(* CODESYS project SPT_Base_Types.library
   Company: Beckhoff Automation LLC
   DefaultNamespace: SPT_BaseTypes
   Version: 3.2.3
   Placeholder: SPT Base Types
   Title: SPT Base Types

Project tree, tasks and I/O mapping:
  libraries: SPT Event Logger, * (Beckhoff Automation LLC); Tc2_EtherCAT, * (Beckhoff Automation GmbH); Tc2_Standard, * (Beckhoff Automation GmbH); Tc2_System, * (Beckhoff Automation GmbH); Tc2_Utilities, * (Beckhoff Automation GmbH); Tc3_EventLogger, * (Beckhoff Automation GmbH); Tc3_JsonXml, * (Beckhoff Automation GmbH); Tc3_PackML_V2, * (Beckhoff Automation GmbH)
  Component Base/
    HMI/
      data type ST_ComponentBase_Command
      data type ST_ComponentBase_Config
      data type ST_ComponentBase_HMI
      data type ST_ComponentBase_Status
    function block FB_ComponentBase [ST]: AllowHMIControl, BlockHMIControl, Reset, CurrentAlarmSeverity, InSimulation, Name, ParentResponseDefinitions, CyclicLogic, CreateEvents, HMICommunication, Initialize, Monitoring, RaiseAlarm, RaiseAlarmWithStrings, RaiseEventWithStrings
  Framework Base/
    function block FB_BaseFB [ST]: Busy, Error, ErrorID, Marker, Trace, TraceWithJson
    function block FB_CyclicFB [ST]: CyclicLogic, InitComplete
  Interfaces/
    interface I_BaseFB: Busy, Error, ErrorID
    interface I_ComponentBase: AllowHMIControl, BlockHMIControl, Reset, CurrentAlarmSeverity, InSimulation, Name, ParentResponseDefinitions
    interface I_CyclicFB: CyclicLogic, InitComplete
    interface I_PackML_BaseModule: CurrentAlarmSeverity, LogModeChanges, LogStateChanges, Name, ParentResponseDefinitions
    interface I_PackML_Control: ChangeMode, ChangeState, CurrentMode, CurrentState, ModeCommand, StateCommand
    interface I_PackML_ExternalController: Control, ModeChanged, StateChanged
  PackML/
    ControlSource/
      function block FB_ControlSource [ST]: CyclicLogic, Control, ModeChanged, StateChanged, Initialize, Registered
      data type ST_PackML_Control
      data type ST_PackML_Control_Simplified
    DUT/
      data type E_AlarmResponse
      data type E_PMLUnitMode
      data type ST_PackML_SubUnitInfoExt
    HMI/
      data type ST_PackMLBaseModule_Command
      data type ST_PackMLBaseModule_Config
      data type ST_PackMLBaseModule_HMI
      data type ST_PackMLBaseModule_Status
    function block FB_PackML_BaseModule [ST]: CyclicLogic, CurrentAlarmSeverity, LogModeChanges, LogStateChanges, Name, ParentResponseDefinitions, ChangeMode, ChangeState, CurrentMode, CurrentState, ModeCommand, StateCommand, AbortImmediate, AbortImmediateError, HoldControlled, HoldImmediate, StopControlled, StopImmediate, SuspendControlled, SuspendImmediate, RaiseAlarmWithStrings, AllowHMIControl, BlockHMIControl, HMICommunication, HMIPermissions, ComponentMonitor, SubModuleMonitor, Aborted, Complete, Execute, Held, Idle, Stopped, Suspended, Undefined, ModeControl, StateControl, Aborting, Clearing, Completing, Holding, Resetting, Starting, Stopping, Suspending, Unholding, Unsuspending, CreateEvents, Initialize, RegisterComponent, RegisterExternalController, RegisterSubmodule, StateComplete
    function block FB_PackML_ModeLogger [ST]
    function block FB_PackML_StateLogger [ST]
  Project Information/
    function F_GetCompany [ST]
    function F_GetTitle [ST]
    function F_GetVersion [ST]
  Tracing/
    function block FB_TraceLog [ST]: AddContext, AddEntry, AddEntryWithJson, FB_init, TracingAllowed
    global variables Tracing
  Version/
    global variables Global_Version
  VISUs/
    visualisation V_MachineModule
    visualisation V_Module
  text list GlobalTextList
  00000000-0000-0000-0000-000000000000|LICENSE
  LICENSE
  global variables Parameters_BaseComponent
  global variables Parameters_PackML_Base
  global variables Parameters_Tracing
*)

// Component Base/HMI/ST_ComponentBase_Command
TYPE ST_ComponentBase_Command :
	STRUCT
		SimulatedOperation : BOOL;
		StandardOperation  : BOOL;
		Reset			   : BOOL;
	END_STRUCT
END_TYPE

// Component Base/HMI/ST_ComponentBase_Config
TYPE ST_ComponentBase_Config :
	STRUCT
		Name : STRING;
	END_STRUCT
END_TYPE

// Component Base/HMI/ST_ComponentBase_HMI
TYPE ST_ComponentBase_HMI :
	STRUCT
		Config	: ST_ComponentBase_Config;
		Command : ST_ComponentBase_Command;
		Status	: ST_ComponentBase_Status;
	END_STRUCT
END_TYPE

// Component Base/HMI/ST_ComponentBase_Status
TYPE ST_ComponentBase_Status :
	STRUCT
		InSimulation		: BOOL;
		Busy				: BOOL;
		Error				: BOOL;
		ErrorID				: UDINT;
		HMIControlAvailable : BOOL; //Set TRUE *FROM PLC* when HMI requests can be processed
	END_STRUCT
END_TYPE

// PackML/ControlSource/ST_PackML_Control
TYPE ST_PackML_Control :
	STRUCT
		CurrentMode		 : E_PMLUnitMode;
		ModeCommand		 : E_PMLUnitMode;
		CurrentState	 : E_PMLState;
		StateCommand	 : E_PMLCommand;
		ModeNames		 : ARRAY[0..31] OF STRING;
		ModeCommandLast	 : E_PMLUnitMode;
		StateCommandLast : E_PMLCommand;
	END_STRUCT
END_TYPE

// PackML/ControlSource/ST_PackML_Control_Simplified
TYPE ST_PackML_Control_Simplified :
	STRUCT
		ResetPermissive		: BOOL;
		StartPermissive		: BOOL;
		StopPermissive		: BOOL;
		ResetPressed AT %I* : BOOL;
		StartPressed AT %I* : BOOL;
		StopPressed	 AT %I* : BOOL;
	END_STRUCT
END_TYPE

// PackML/DUT/E_AlarmResponse
//! @summary Defines the reaction behavior to a fault
{attribute 'qualified_only'}
{attribute 'strict'}
TYPE E_AlarmResponse : (
		Abort_ImmediateError,
		Abort_Immediate,
		Stop_Immediate,
		Stop_Controlled,
		Hold_Immediate,
		Hold_Controlled,
		Suspend_Immediate,
		Suspend_Controlled,
		NoResponse
	);
END_TYPE

// PackML/DUT/E_PMLUnitMode
//! @summary Defines the allowable PackML modes  
TYPE E_PMLUnitMode : (
		ePMLUnitMode_Invalid	 := 0,
		ePMLUnitMode_Production	 := 1,
		ePMLUnitMode_Maintenance := 2,
		ePMLUnitMode_Manual		 := 3,
		ePMLUnitMode_UserMode1	 := 4,
		ePMLUnitMode_UserMode2	 := 5,
		ePMLUnitMode_UserMode3	 := 6,
		ePMLUnitMode_UserMode4	 := 7,
		ePMLUnitMode_UserMode5	 := 8,
		ePMLUnitMode_UserMode6	 := 9,
		ePMLUnitMode_UserMode7	 := 10,
		ePMLUnitMode_UserMode8	 := 11,
		ePMLUnitMode_UserMode9	 := 12,
		ePMLUnitMode_UserMode10	 := 13,
		ePMLUnitMode_UserMode11	 := 14,
		ePMLUnitMode_UserMode12	 := 15,
		ePMLUnitMode_UserMode13	 := 16,
		ePMLUnitMode_UserMode14	 := 17,
		ePMLUnitMode_UserMode15	 := 18,
		ePMLUnitMode_UserMode16	 := 19,
		ePMLUnitMode_UserMode17	 := 20,
		ePMLUnitMode_UserMode18	 := 21,
		ePMLUnitMode_UserMode19	 := 22,
		ePMLUnitMode_UserMode20	 := 23,
		ePMLUnitMode_UserMode21	 := 24,
		ePMLUnitMode_UserMode22	 := 25,
		ePMLUnitMode_UserMode23	 := 26,
		ePMLUnitMode_UserMode24	 := 27,
		ePMLUnitMode_UserMode25	 := 28,
		ePMLUnitMode_UserMode26	 := 29,
		ePMLUnitMode_UserMode27	 := 30,
		ePMLUnitMode_UserMode28	 := 31
	) DINT;
END_TYPE

// PackML/DUT/ST_PackML_SubUnitInfoExt
TYPE ST_PackML_SubUnitInfoExt EXTENDS ST_PMLSubUnitInfo : //Extended Struct of ST_PMLSubUnitInfo
	STRUCT
		ModuleID		: DINT;	  //Machine ID for messaging and Identification
		ModuleName		: STRING; //Human readable machine name for messaging
		UnitModeCurrent : E_PMLProtectedUnitMode;
		ActiveAlarm		: BOOL;
	END_STRUCT
END_TYPE

// PackML/HMI/ST_PackMLBaseModule_Command
TYPE ST_PackMLBaseModule_Command :
	STRUCT
		Mode			   : E_PMLUnitMode				:= Parameters_PackML_Base.UNIT_MODE_DEFAULT;
		State			   : Tc3_PackML_V2.E_PMLCommand := Parameters_PackML_Base.UNIT_STATE_DEFAULT;
		ActivateStateLog   : BOOL; //HMI requests to enable the module
		DeactivateStateLog : BOOL; //HMI requests to disable the module
		ActivateModeLog	   : BOOL; //HMI requests to enable the module
		DeactivatModeLog   : BOOL; //HMI requests to disable the module
	END_STRUCT
END_TYPE

// PackML/HMI/ST_PackMLBaseModule_Config
TYPE ST_PackMLBaseModule_Config :
	STRUCT
		Name			: STRING;		//Human-readable module name for user-side messaging
		LogStateChanges : BOOL := TRUE; //Toggle to permit or suppress state change logging (Should be tied to HMI setting to optionally reduce event logger clutter)
		LogModeChanges	: BOOL := TRUE; //Toggle to permit or suppress state change logging (Should be tied to HMI setting to optionally reduce event logger clutter)
		ModeNames		: ARRAY[0..31] OF STRING;
	END_STRUCT
END_TYPE

// PackML/HMI/ST_PackMLBaseModule_HMI
TYPE ST_PackMLBaseModule_HMI :
	STRUCT
		Config	: ST_PackMLBaseModule_Config;
		Command : ST_PackMLBaseModule_Command;
		Status	: ST_PackMLBaseModule_Status;
	END_STRUCT
END_TYPE

// PackML/HMI/ST_PackMLBaseModule_Status
TYPE ST_PackMLBaseModule_Status :
	STRUCT
		Busy				: BOOL;
		Error				: BOOL;
		ErrorID				: UDINT;
		Mode				: E_PMLUnitMode;
		State				: Tc3_PackML_V2.E_PMLState;
		HMIControlAvailable : BOOL;
	END_STRUCT
END_TYPE

// Tracing/Tracing
{attribute 'qualified_only'}
VAR_GLOBAL
	GlobalTraceLog : FB_TraceLog;
END_VAR

// Version/Global_Version
{attribute 'TcGenerated'}
{attribute 'no-analysis'}
{attribute 'linkalways'}
// This function has been automatically generated from the project information.
VAR_GLOBAL CONSTANT
	{attribute 'const_non_replaced'}
	stLibVersion_SPT_Base_Types : ST_LibVersion := (iMajor := 3, iMinor := 2, iBuild := 3, iRevision := 0, nFlags := 1, sVersion := '3.2.3');
END_VAR

// Parameters_BaseComponent
{attribute 'qualified_only'}
VAR_GLOBAL CONSTANT
	COMPONENT_BASE_ALARM_COUNT : UINT := 2;
END_VAR

// Parameters_PackML_Base
{attribute 'qualified_only'}
VAR_GLOBAL CONSTANT
	MAX_NO_OF_SUBMODULES		   : UDINT						:= 20;
	MAX_NO_OF_COMPONENTS		   : UDINT						:= 32;
	MAX_NO_OF_EXTERNAL_CONTROLLERS : UDINT						:= 10;
	UNIT_MODE_DEFAULT			   : E_PMLUnitMode				:= E_PMLUnitMode.ePMLUnitMode_Production;
	UNIT_STATE_DEFAULT			   : Tc3_PackML_V2.E_PMLCommand := E_PMLCommand.ePMLCommand_Abort;
END_VAR

// Parameters_Tracing
{attribute 'qualified_only'}
VAR_GLOBAL CONSTANT
	TRACING_ENABLED						: BOOL	:= TRUE;
	MAX_LOG_ENTRIES_PER_SCAN			: UDINT := 100;
	ALLOW_DUPLICATE_SEQUENTIAL_MESSAGES : BOOL	:= FALSE;
END_VAR

// Component Base/FB_ComponentBase
//! @summary Basic framework of a component
FUNCTION_BLOCK ABSTRACT FB_ComponentBase EXTENDS FB_CyclicFB IMPLEMENTS I_ComponentBase
VAR
	//I_BasicComponent internal property variables
	_CurrentAlarmSeverity			: TcEventSeverity;
	_Name							: STRING; //String name of the component
	_ParentFaultResponseDefinitions : ARRAY[0..4] OF E_AlarmResponse
		:= [E_AlarmResponse.NoResponse, E_AlarmResponse.NoResponse, E_AlarmResponse.NoResponse, E_AlarmResponse.Abort_ImmediateError, E_AlarmResponse.Abort_ImmediateError];
	_Simulate : BOOL; //TRUE disables all hardware I/O and simulates input and output behavior

	//Alarming
	ComponentBaseAlarms : ARRAY[1..Parameters_BaseComponent.COMPONENT_BASE_ALARM_COUNT] OF FB_TcAlarm;

	//HMI Monitoring and control structure
	ComponentBase_HMI			: ST_ComponentBase_HMI;
	HMICommand_RT				: R_TRIG;
	HMICommandActive_Base		: BOOL;
	HMICommandActive_Descendant : BOOL;
END_VAR

//! @summary Sets permissive bit to allow HMI control of component functions
METHOD PUBLIC AllowHMIControl

//! @description This method is called as required by the parent module of this component
ComponentBase_HMI.Status.HMIControlAvailable := TRUE;
END_METHOD

//! @summary Clears permissive bit to allow HMI control of component functions
METHOD PUBLIC BlockHMIControl

//! @description This method is called as required by the parent module of this component
ComponentBase_HMI.Status.HMIControlAvailable := FALSE;
END_METHOD

//! @summary Clears error flags and error IDs for this component
METHOD PUBLIC Reset : BOOL
//This may or may not be called depending on the component type 

//which derives FB_ComponentBase
F_ClearAllEventsInClass(ComponentBaseAlarms);
Reset := TRUE;
END_METHOD

//! @summary Returns the current alarm severity for this component
PROPERTY CurrentAlarmSeverity : TcEventSeverity
GET
CurrentAlarmSeverity := _CurrentAlarmSeverity;
END_GET
END_PROPERTY

//! @summary Enable/Disable simulation logic for this component
PROPERTY InSimulation : BOOL
GET
InSimulation := _Simulate;
END_GET
SET
_Simulate := InSimulation;
END_SET
END_PROPERTY

//! @summary Get/Set this component's name
PROPERTY Name : STRING
GET
Name := _Name;
END_GET
SET
_Name := Name;
END_SET
END_PROPERTY

PROPERTY ParentResponseDefinitions : ARRAY[0..4] OF E_AlarmResponse
GET
ParentResponseDefinitions[TcEventSeverity.Verbose]	:= _ParentFaultResponseDefinitions[TcEventSeverity.Verbose];
ParentResponseDefinitions[TcEventSeverity.Info]		:= _ParentFaultResponseDefinitions[TcEventSeverity.Info];
ParentResponseDefinitions[TcEventSeverity.Warning]	:= _ParentFaultResponseDefinitions[TcEventSeverity.Warning];
ParentResponseDefinitions[TcEventSeverity.Error]	:= _ParentFaultResponseDefinitions[TcEventSeverity.Error];
ParentResponseDefinitions[TcEventSeverity.Critical] := _ParentFaultResponseDefinitions[TcEventSeverity.Critical];
END_GET
SET
_ParentFaultResponseDefinitions[TcEventSeverity.Verbose]  := ParentResponseDefinitions[TcEventSeverity.Verbose];
_ParentFaultResponseDefinitions[TcEventSeverity.Info]	  := ParentResponseDefinitions[TcEventSeverity.Info];
_ParentFaultResponseDefinitions[TcEventSeverity.Warning]  := ParentResponseDefinitions[TcEventSeverity.Warning];
_ParentFaultResponseDefinitions[TcEventSeverity.Error]	  := ParentResponseDefinitions[TcEventSeverity.Error];
_ParentFaultResponseDefinitions[TcEventSeverity.Critical] := ParentResponseDefinitions[TcEventSeverity.Critical];
END_SET
END_PROPERTY

//! @summary This method serves as the entry point for all underlying FB logic
METHOD PUBLIC CyclicLogic

//! @description This method should be called cyclically by descendant function blocks by invoking <c>SUPER^.CyclicLogic()</c>.  Alternatively, the contents of this method could be reimplemented entirely in which case a call to this method would not be necessary.
IF NOT _InitComplete THEN
	_InitComplete := Initialize();
	RETURN;
END_IF

Monitoring();		//Constant error and status monitoring
HMICommunication(); //Keeps the HMI data up to date, and processes requests from the HMI for this component
END_METHOD

//! @summary Initializes event function blocks using this components's name
{attribute 'call_after_online_change_slot' := '<slot>'}
METHOD PROTECTED CreateEvents

//! @description This method is called by <c>Initialize()</c> as required
F_CreateAllEventsInClass(Alarms		:= ComponentBaseAlarms,
						 ClassSize	:= SIZEOF(TC_EVENTS.ComponentBase),
						 pInitEvent := ADR(TC_EVENTS.ComponentBase.InitReferenceEvent),
						 Prefix		:= _Name);
END_METHOD

//! @summary Provides interlocks for HMI control and updates HMI status information for this component
METHOD PROTECTED HMICommunication

//! @description This method is called cyclically by <c>CyclicLogic()</c>
//Extend this method in extended FBs to communicate specific implementation data

//Process HMI requests
HMICommand_RT(CLK := (ComponentBase_HMI.Status.HMIControlAvailable AND NOT HMICommandActive_Descendant) AND
					 (ComponentBase_HMI.Command.Reset XOR ComponentBase_HMI.Command.SimulatedOperation XOR ComponentBase_HMI.Command.StandardOperation));

//Desendant components should observe this to interlock HMI commands
HMICommandActive_Base :=
	ComponentBase_HMI.Status.HMIControlAvailable AND (ComponentBase_HMI.Command.Reset OR ComponentBase_HMI.Command.SimulatedOperation OR ComponentBase_HMI.Command.StandardOperation);

IF HMICommand_RT.Q THEN
	IF ComponentBase_HMI.Command.Reset THEN
		Reset();
	END_IF

	IF ComponentBase_HMI.Command.SimulatedOperation THEN
		_Simulate := TRUE;
	END_IF

	IF ComponentBase_HMI.Command.StandardOperation THEN
		_Simulate := FALSE;
	END_IF
END_IF

//Update HMI status info
ComponentBase_HMI.Config.Name		  := _Name;
ComponentBase_HMI.Status.Busy		  := _Busy;
ComponentBase_HMI.Status.Error		  := _Error;
ComponentBase_HMI.Status.InSimulation := _Simulate;
ComponentBase_HMI.Status.ErrorID	  := _ErrorID;
END_METHOD

//! @summary Basic component initialization logic
METHOD PROTECTED Initialize : BOOL;

//! @description This method is called by <c>CyclicLogic()</c> as required
//Extend initialize as needed in extended FBs
CreateEvents();
Initialize := TRUE;
END_METHOD

//! Provides basic error detection and event handling for this component
METHOD PROTECTED Monitoring

(*! @descriptionThis method is called cyclically by <c>CyclicLogic()</c>*)
//Extend from extended FB with monitoring logic
IF NOT ComponentBaseAlarms[E_ComponentBase.SimulationWarning].bRaised AND _Simulate THEN
	ComponentBaseAlarms[E_ComponentBase.SimulationWarning].Raise(0);
ELSIF ComponentBaseAlarms[E_ComponentBase.SimulationWarning].bRaised AND NOT _Simulate THEN
	ComponentBaseAlarms[E_ComponentBase.SimulationWarning].Clear(0, 0);
END_IF

_CurrentAlarmSeverity := TcEventSeverity.Verbose;
_CurrentAlarmSeverity := F_GetMaxSeverityRaised(Alarms := ComponentBaseAlarms, CurrentSeverity := _CurrentAlarmSeverity);
END_METHOD

//! @summary Raise an alarm, passing the faulted FB's error ID as a paramter
METHOD PROTECTED RaiseAlarm
VAR_IN_OUT
	Alarm : FB_TcAlarm;
END_VAR
F_RaiseAlarm(Alarm := Alarm);
END_METHOD

//! @summary Raises an alarm and passes string arguments as parameters for extra fault context/info
METHOD PROTECTED RaiseAlarmWithStrings
VAR_IN_OUT
	Alarm : FB_TcAlarm; //! Alarm to be raised
END_VAR

VAR_INPUT
	String_1 : STRING; //! First string parameter (The Name of this component will be applied first automatically)
	String_2 : STRING; //! Second string parameter
END_VAR
F_RaiseAlarmWithStringsAndFlags(Alarm	  := Alarm,
								ErrorFlag := _Error,
								ErrorID	  := _ErrorID,
								String_1  := _Name,
								String_2  := String_1,
								String_3  := String_2);
END_METHOD

//! @summary Raises an alarm and passes string arguments as parameters for extra fault context/info
METHOD PROTECTED RaiseEventWithStrings
VAR_IN_OUT
	Alarm : FB_TcAlarm; //! Alarm to be raised
END_VAR

VAR_INPUT
	String_1 : STRING; //! First string parameter (The Name of this component will be applied first automatically)
	String_2 : STRING; //! Second string parameter
END_VAR
F_RaiseAlarmWithStringParameters(Alarm	  := Alarm,
								 String_1 := _Name,
								 String_2 := String_1,
								 String_3 := String_2);
END_METHOD

END_FUNCTION_BLOCK

// Framework Base/FB_CyclicFB
FUNCTION_BLOCK ABSTRACT FB_CyclicFB EXTENDS FB_BaseFB IMPLEMENTS I_CyclicFB
VAR
	_InitComplete : BOOL;
END_VAR

// Derivatives of FB_CyclicFB should *NOT* have code in the function block body

// Use CyclicLogic() instead

METHOD PUBLIC ABSTRACT CyclicLogic
VAR_INPUT
END_VAR
END_METHOD

PROPERTY InitComplete : BOOL
GET
InitComplete := _InitComplete;
END_GET
END_PROPERTY

END_FUNCTION_BLOCK

// Framework Base/FB_BaseFB
{attribute 'reflection'}
FUNCTION_BLOCK ABSTRACT FB_BaseFB IMPLEMENTS I_BaseFB
VAR
	{attribute 'instance-path'}
	{attribute 'noinit'}
	InstancePath : STRING;
END_VAR

// I_BaseFB
VAR
	_Busy	 : BOOL := TRUE;
	_Error	 : BOOL;
	_ErrorID : UDINT;
END_VAR

// Derivatives of FB_BaseFB can have code in the function block body

PROPERTY Busy : BOOL
GET
Busy := _Busy;
END_GET
END_PROPERTY

PROPERTY Error : BOOL
GET
Error := _Error;
END_GET
END_PROPERTY

PROPERTY ErrorID : UDINT
GET
ErrorID := _ErrorID;
END_GET
END_PROPERTY

METHOD PUBLIC Marker
VAR_INPUT
	Message : T_MaxString;
END_VAR
Tracing.GlobalTraceLog.AddEntry(InstancePath, Message, 1);
END_METHOD

METHOD PUBLIC Trace
VAR_INPUT
	Message : T_MaxString;
END_VAR
Tracing.GlobalTraceLog.AddEntry(InstancePath, Message, 0);
END_METHOD

METHOD PUBLIC TraceWithJson
VAR_INPUT
	Message : T_MaxString;
	Json	: T_MaxString;
END_VAR
Tracing.GlobalTraceLog.AddEntryWithJson(InstancePath,
										Message,
										0,
										Json);
END_METHOD

END_FUNCTION_BLOCK

// Interfaces/I_BaseFB
INTERFACE I_BaseFB EXTENDS __SYSTEM.IQueryInterface

PROPERTY Busy : BOOL
GET
END_GET
END_PROPERTY

PROPERTY Error : BOOL
GET
END_GET
END_PROPERTY

PROPERTY ErrorID : UDINT;
GET
END_GET
END_PROPERTY

END_INTERFACE

// Interfaces/I_CyclicFB
INTERFACE I_CyclicFB EXTENDS I_BaseFB

METHOD CyclicLogic
VAR_INPUT
END_VAR
END_METHOD

PROPERTY InitComplete : BOOL
GET
END_GET
END_PROPERTY

END_INTERFACE

// Interfaces/I_ComponentBase
INTERFACE I_ComponentBase EXTENDS I_CyclicFB

METHOD PUBLIC AllowHMIControl
VAR_INPUT
END_VAR
END_METHOD

METHOD PUBLIC BlockHMIControl
VAR_INPUT
END_VAR
END_METHOD

METHOD PUBLIC Reset : BOOL
END_METHOD

PROPERTY CurrentAlarmSeverity : TcEventSeverity
GET
END_GET
END_PROPERTY

PROPERTY InSimulation : BOOL
GET
END_GET
SET
END_SET
END_PROPERTY

PROPERTY Name : STRING
GET
END_GET
SET
END_SET
END_PROPERTY

PROPERTY ParentResponseDefinitions : ARRAY[0..4] OF E_AlarmResponse
GET
END_GET
SET
END_SET
END_PROPERTY

END_INTERFACE

// Interfaces/I_PackML_BaseModule
INTERFACE I_PackML_BaseModule EXTENDS I_CyclicFB, I_PackML_Control

PROPERTY CurrentAlarmSeverity : TcEventSeverity
GET
END_GET
END_PROPERTY

PROPERTY LogModeChanges : BOOL
GET
END_GET
SET
END_SET
END_PROPERTY

PROPERTY LogStateChanges : BOOL
GET
END_GET
SET
END_SET
END_PROPERTY

PROPERTY Name : STRING
GET
END_GET
SET
END_SET
END_PROPERTY

PROPERTY ParentResponseDefinitions : ARRAY[0..4] OF E_AlarmResponse
GET
END_GET
SET
END_SET
END_PROPERTY

END_INTERFACE

// Interfaces/I_PackML_Control
INTERFACE I_PackML_Control

METHOD ChangeMode
VAR_INPUT
	Mode : E_PMLUnitMode;
END_VAR
END_METHOD

METHOD ChangeState
VAR_INPUT
	State : E_PMLCommand;
END_VAR
END_METHOD

PROPERTY CurrentMode : E_PMLUnitMode
GET
END_GET
END_PROPERTY

PROPERTY CurrentState : E_PMLState
GET
END_GET
END_PROPERTY

PROPERTY ModeCommand : DINT
GET
END_GET
SET
END_SET
END_PROPERTY

PROPERTY StateCommand : E_PMLCommand
GET
END_GET
SET
END_SET
END_PROPERTY

END_INTERFACE

// Interfaces/I_PackML_ExternalController
INTERFACE I_PackML_ExternalController

PROPERTY Control : I_PackML_Control
SET
END_SET
END_PROPERTY

METHOD ModeChanged
VAR_INPUT
	NewMode : E_PMLUnitMode;
END_VAR
END_METHOD

METHOD StateChanged
VAR_INPUT
	NewState : E_PMLCommand;
END_VAR
END_METHOD

END_INTERFACE

// PackML/ControlSource/FB_ControlSource
FUNCTION_BLOCK FB_ControlSource EXTENDS FB_CyclicFB IMPLEMENTS I_PackML_ExternalController
VAR
	ipModule				  : I_PackML_Control;
	MainPMLControl_Simplified : ST_PackML_Control_Simplified;
	MainPMLControl_Standard	  : ST_PackML_Control;
	R_HMICommand			  : R_TRIG;
END_VAR

METHOD CyclicLogic
VAR
	i : UDINT;
END_VAR
IF NOT _InitComplete THEN
	_InitComplete := Initialize();
	RETURN;
END_IF

//Copy the module to the local mode and state
MainPMLControl_Standard.CurrentMode	 := ipModule.CurrentMode;
MainPMLControl_Standard.CurrentState := ipModule.CurrentState;
FOR i := 1 TO 5 DO
	MainPMLControl_Standard.ModeNames[i] := F_UnitModeToString(TO_DINT(i));
END_FOR

//Process requests
R_HMICommand(CLK := (MainPMLControl_Simplified.ResetPressed XOR MainPMLControl_Simplified.StartPressed XOR MainPMLControl_Simplified.StopPressed) XOR
					(MainPMLControl_Standard.StateCommand <> E_PMLCommand.ePMLCommand_Undefined AND MainPMLControl_Standard.StateCommandLast <> MainPMLControl_Standard.StateCommand) XOR
					(MainPMLControl_Standard.ModeCommandLast <> MainPMLControl_Standard.ModeCommand));

IF R_HMICommand.Q THEN
	MainPMLControl_Standard.ModeCommandLast	 := MainPMLControl_Standard.ModeCommand;
	MainPMLControl_Standard.StateCommandLast := MainPMLControl_Standard.StateCommand;
	IF MainPMLControl_Simplified.ResetPressed AND MainPMLControl_Simplified.ResetPermissive AND MainPMLControl_Standard.CurrentState = E_PMLState.ePMLState_Aborted THEN
		ipModule.ChangeState(Tc3_PackML_V2.E_PMLCommand.ePMLCommand_Clear);
	ELSIF MainPMLControl_Simplified.ResetPressed AND MainPMLControl_Simplified.ResetPermissive THEN
		ipModule.ChangeState(Tc3_PackML_V2.E_PMLCommand.ePMLCommand_Reset);
	ELSIF MainPMLControl_Simplified.StartPressed AND MainPMLControl_Simplified.StartPermissive THEN
		IF MainPMLControl_Standard.CurrentState = Tc3_PackML_V2.E_PMLState.ePMLState_Idle THEN
			ipModule.ChangeState(Tc3_PackML_V2.E_PMLCommand.ePMLCommand_Start);
		ELSIF MainPMLControl_Standard.CurrentState = Tc3_PackML_V2.E_PMLState.ePMLState_Held THEN
			ipModule.ChangeState(Tc3_PackML_V2.E_PMLCommand.ePMLCommand_Unhold);
		END_IF
	ELSIF MainPMLControl_Simplified.StopPressed AND MainPMLControl_Simplified.StopPermissive THEN
		ipModule.ChangeState(Tc3_PackML_V2.E_PMLCommand.ePMLCommand_Stop);
	ELSIF ipModule.StateCommand <> MainPMLControl_Standard.StateCommand THEN
		ipModule.StateCommand := MainPMLControl_Standard.StateCommand;
	ELSIF ipModule.ModeCommand <> MainPMLControl_Standard.ModeCommand THEN
		ipModule.ModeCommand := MainPMLControl_Standard.ModeCommand;
	END_IF
END_IF

//Set the permissives for each button
MainPMLControl_Simplified.StartPermissive :=
	MainPMLControl_Standard.CurrentState = Tc3_PackML_V2.E_PMLState.ePMLState_Idle OR MainPMLControl_Standard.CurrentState = Tc3_PackML_V2.E_PMLState.ePMLState_Held;

MainPMLControl_Simplified.StopPermissive :=
	(MainPMLControl_Standard.CurrentState <> Tc3_PackML_V2.E_PMLState.ePMLState_Stopped AND MainPMLControl_Standard.CurrentState <> Tc3_PackML_V2.E_PMLState.ePMLState_Clearing AND
	 MainPMLControl_Standard.CurrentState <> Tc3_PackML_V2.E_PMLState.ePMLState_Aborted AND MainPMLControl_Standard.CurrentState <> Tc3_PackML_V2.E_PMLState.ePMLState_Aborting AND
	 MainPMLControl_Standard.CurrentState <> Tc3_PackML_V2.E_PMLState.ePMLState_Idle AND MainPMLControl_Standard.CurrentState <> Tc3_PackML_V2.E_PMLState.ePMLState_Undefined);

MainPMLControl_Simplified.ResetPermissive :=
	MainPMLControl_Standard.CurrentState = Tc3_PackML_V2.E_PMLState.ePMLState_Complete OR MainPMLControl_Standard.CurrentState = Tc3_PackML_V2.E_PMLState.ePMLState_Stopped OR
	MainPMLControl_Standard.CurrentState = Tc3_PackML_V2.E_PMLState.ePMLState_Aborted;
END_METHOD

PROPERTY Control : I_PackML_Control
SET
ipModule := Control;
END_SET
END_PROPERTY

METHOD FINAL ModeChanged
VAR_INPUT
	NewMode : E_PMLUnitMode;
END_VAR
MainPMLControl_Standard.ModeCommand := NewMode;
END_METHOD

METHOD FINAL StateChanged
VAR_INPUT
	NewState : E_PMLCommand;
END_VAR
MainPMLControl_Standard.StateCommand := NewState;
END_METHOD

METHOD FINAL Initialize : BOOL
IF Registered THEN
	Initialize := TRUE;
END_IF
END_METHOD

PROPERTY Registered : BOOL
GET
Registered := ipModule <> 0;
END_GET
END_PROPERTY

END_FUNCTION_BLOCK

// PackML/FB_PackML_BaseModule
FUNCTION_BLOCK ABSTRACT FB_PackML_BaseModule EXTENDS FB_CyclicFB IMPLEMENTS I_PackML_BaseModule, I_PackML_Control
	//I_PMLControl
VAR
	_CurrentMode	: E_PMLUnitMode; //Current UnitMode of the module	
	_CommandedMode	: E_PMLUnitMode; //Current Commanded UnitMode of the module
	_CurrentState	: Tc3_PackML_V2.E_PMLState;
	_CommandedState : Tc3_PackML_V2.E_PMLCommand;
END_VAR

//I_PMLModuleBase
VAR
	_CurrentAlarmSeverity			: TcEventSeverity;
	_LogModeChanges					: BOOL := TRUE;	 //Toggle to permit or suppress state change logging (Should be tied to HMI setting to optionally reduce event logger clutter)
	_LogStateChanges				: BOOL := FALSE; //Toggle to permit or suppress state change logging (Should be tied to HMI setting to optionally reduce event logger clutter)
	_Name							: STRING;		 //Human-readable module name for user-side messaging
	_ParentFaultResponseDefinitions : ARRAY[0..4] OF E_AlarmResponse
		:= [E_AlarmResponse.NoResponse, E_AlarmResponse.NoResponse, E_AlarmResponse.NoResponse, E_AlarmResponse.Abort_ImmediateError, E_AlarmResponse.Abort_ImmediateError];
END_VAR

VAR
	ModeManager						  : PML_UnitModeManager;		//Manages operating mode transitions and rules
	StateMachine					  : PML_StateMachine;			//Manages PackML state transitions
	CustomModes						  : PML_UnitModeConfig;			//Used to define custom machine modes if desired
	PMLStateLogger					  : FB_PackML_StateLogger;		//Logs PackML state changes
	PMLModeLogger					  : FB_PackML_ModeLogger;		//Logs PackML Mode changes	
	PackMLBaseModule_HMI			  : ST_PackMLBaseModule_HMI;	//Handles status and control communications with the HMI
	PMLSubModuleInfoRef				  : ST_PMLSubUnitInfoRef;		// Reference to the subunit information, used by the state machine
	LastModeCommand					  : E_PMLUnitMode;				//Previous received PackML mode command
	LastMode						  : DINT;						//Last PackML mode 	
	LastState						  : Tc3_PackML_V2.E_PMLState;	//Last cycle PackML state
	StateTasksComplete				  : BOOL := FALSE;				//All tasks to be performed at this program level are complete
	NoStateTasksToComplete			  : BOOL := TRUE;				//Indicates whether this stateneeds to perform tasks other than commanding its children
	PackMLAlarms					  : ARRAY[1..48] OF FB_TcAlarm; //Array of alarms for PackML state and mode changes that exist in any PackML enabled module
	BaseAlarms						  : ARRAY[1..32] OF FB_TcAlarm; //Array of alarms for general module Alarms				
	ipSubModules					  : ARRAY[1..Parameters_PackML_Base.MAX_NO_OF_SUBMODULES] OF I_PackML_BaseModule;
	PMLSubModuleInfo				  : ARRAY[1..Parameters_PackML_Base.MAX_NO_OF_SUBMODULES] OF ST_PMLSubUnitInfo;
	NumberOfSubModules				  : UDINT := 0; //calculated number of instantiated sub modules
	ipComponents					  : ARRAY[1..Parameters_PackML_Base.MAX_NO_OF_COMPONENTS] OF I_ComponentBase;
	NumberOfComponents				  : UDINT := 0; //calculated number of instantiated components
	ModeNames						  : ARRAY[0..31] OF STRING;
	ipExternalControllers			  : ARRAY[1..Parameters_PackML_Base.MAX_NO_OF_EXTERNAL_CONTROLLERS] OF I_PackML_ExternalController;
	ReachedInitialDefaultStateAndMode : BOOL;
	ModeChangeRequested				  : BOOL;
	SequenceState					  : UDINT;
	DescendantSequenceState			  : UDINT;
	HMICommand_RT					  : R_TRIG;
	HMICommandActive_Base			  : BOOL;
	HMICommandActive_Descendant		  : BOOL;
END_VAR

//*********************************************************

// !!!!! Code implementation only in CyclicLogic() method !!!!! 

//*********************************************************

//! @summary This method serves as the entry point for all underlying FB logic

//! @description This method should be called cyclically by descendant function blocks by invoking <c>SUPER^.CyclicLogic()</c>.  Alternatively, the contents of this method could be reimplemented entirely in which case a call to this method would not be necessary.
METHOD PUBLIC CyclicLogic
VAR
	i : UDINT;
END_VAR
//*********************************************************

//If you are about to write actual machine implementation code, note that implementation code should exist within an implementation machine module block that extends this machine module base!

//*********************************************************

// Descendents of this FB which override this methods should

// use SUPER^.Initialize()
IF NOT _InitComplete THEN
	_InitComplete := Initialize();
	RETURN;
END_IF

// Inhibit mode & state errors until startup is complete
IF NOT ReachedInitialDefaultStateAndMode AND _CurrentState = E_PMLState.ePMLState_Aborted AND _CurrentMode = Parameters_PackML_Base.UNIT_MODE_DEFAULT THEN
	ReachedInitialDefaultStateAndMode := TRUE;
END_IF

// Call this module's subunits, if any are defined
FOR i := 1 TO NumberOfSubModules DO
	IF ipSubModules[i] <> 0 THEN
		ipSubModules[i].CyclicLogic();
		PMLSubModuleInfo[i].eState := ipSubModules[i].CurrentState; //Reflect the state of the subunits to the state machine of the module		
	END_IF
END_FOR

FOR i := 1 TO NumberOfComponents DO
	IF ipComponents[i] <> 0 THEN
		ipComponents[i].CyclicLogic();
	END_IF
END_FOR

//Handle HMI communications--this must happen before state control!!
HMICommunication();

// Mode control loop of the module
ModeControl();

// State control loop of the module
StateControl();

//VISUCommunication();

//ExternalControl();
SubModuleMonitor();
ComponentMonitor();
HMIPermissions();
_CurrentAlarmSeverity := TcEventSeverity.Verbose;
_CurrentAlarmSeverity := F_GetMaxSeverityRaised(Alarms := PackMLAlarms, CurrentSeverity := _CurrentAlarmSeverity);
_CurrentAlarmSeverity := F_GetMaxSeverityRaised(Alarms := BaseAlarms, CurrentSeverity := _CurrentAlarmSeverity);
END_METHOD

//! @summary Returns the highest severity of any event(s) currently raised 
PROPERTY CurrentAlarmSeverity : TcEventSeverity
GET
CurrentAlarmSeverity := _CurrentAlarmSeverity;
END_GET
END_PROPERTY

//! @summary Enable/Disable logging of mode changes
PROPERTY LogModeChanges : BOOL
GET
LogModeChanges := _LogModeChanges;
END_GET
SET
_LogModeChanges := LogModeChanges;
END_SET
END_PROPERTY

//! @summary Enable/Disable logging of state changes
PROPERTY LogStateChanges : BOOL
GET
LogStateChanges := _LogStateChanges;
END_GET
SET
_LogStateChanges := LogStateChanges;
END_SET
END_PROPERTY

//! @summary Get/Set the name of this module
PROPERTY Name : STRING
GET
Name := _Name;
END_GET
SET
_Name := Name;
END_SET
END_PROPERTY

//! @summary TODO: does this do anything?
PROPERTY ParentResponseDefinitions : ARRAY[0..4] OF E_AlarmResponse
GET
ParentResponseDefinitions[TcEventSeverity.Verbose]	:= _ParentFaultResponseDefinitions[TcEventSeverity.Verbose];
ParentResponseDefinitions[TcEventSeverity.Info]		:= _ParentFaultResponseDefinitions[TcEventSeverity.Info];
ParentResponseDefinitions[TcEventSeverity.Warning]	:= _ParentFaultResponseDefinitions[TcEventSeverity.Warning];
ParentResponseDefinitions[TcEventSeverity.Error]	:= _ParentFaultResponseDefinitions[TcEventSeverity.Error];
ParentResponseDefinitions[TcEventSeverity.Critical] := _ParentFaultResponseDefinitions[TcEventSeverity.Critical];
END_GET
SET
_ParentFaultResponseDefinitions[TcEventSeverity.Verbose]  := ParentResponseDefinitions[TcEventSeverity.Verbose];
_ParentFaultResponseDefinitions[TcEventSeverity.Info]	  := ParentResponseDefinitions[TcEventSeverity.Info];
_ParentFaultResponseDefinitions[TcEventSeverity.Warning]  := ParentResponseDefinitions[TcEventSeverity.Warning];
_ParentFaultResponseDefinitions[TcEventSeverity.Error]	  := ParentResponseDefinitions[TcEventSeverity.Error];
_ParentFaultResponseDefinitions[TcEventSeverity.Critical] := ParentResponseDefinitions[TcEventSeverity.Critical];
END_SET
END_PROPERTY

METHOD ChangeMode
VAR_INPUT
	Mode : E_PMLUnitMode;
END_VAR
IF Mode <> _CommandedMode THEN
	ModeCommand := Mode;
END_IF
END_METHOD

METHOD ChangeState
VAR_INPUT
	State : E_PMLCommand;
END_VAR
IF State <> _CommandedState THEN
	StateCommand := State;
END_IF
END_METHOD

//! @summary Returns the current PackML mode of this module
PROPERTY CurrentMode : E_PMLUnitMode
GET
CurrentMode := _CurrentMode;
END_GET
END_PROPERTY

//! @summary Returns current PackML state of this module
PROPERTY CurrentState : Tc3_PackML_V2.E_PMLState
GET
CurrentState := _CurrentState;
END_GET
END_PROPERTY

//! @summary Sets the requested PackML Mode
PROPERTY ModeCommand : DINT
GET
ModeCommand := _CommandedMode;
END_GET
SET
VAR
	i : UDINT;
END_VAR
IF ModeCommand <> _CommandedMode THEN
	_CommandedMode					  := ModeCommand;
	PackMLBaseModule_HMI.Command.Mode := ModeCommand;

	//Notify external controllers that state has changed	
	FOR i := 1 TO Parameters_PackML_Base.MAX_NO_OF_EXTERNAL_CONTROLLERS DO
		IF ipExternalControllers[i] <> 0 THEN
			ipExternalControllers[i].ModeChanged(_CommandedMode);
		END_IF
	END_FOR

	//ModeChangeRequested := TRUE;
END_IF
END_SET
END_PROPERTY

//! @summary Sets the requested PackML state
PROPERTY StateCommand : Tc3_PackML_V2.E_PMLCommand
GET
StateCommand := _CommandedState;
END_GET
SET
VAR
	i : UDINT;
END_VAR
IF _CurrentMode <> E_PMLUnitMode.ePMLUnitMode_Invalid AND _CurrentState <> E_PMLState.ePMLState_Undefined THEN
	_CommandedState					   := StateCommand;
	PackMLBaseModule_HMI.Command.State := StateCommand;

	//Notify external controllers that state has changed
	FOR i := 1 TO Parameters_PackML_Base.MAX_NO_OF_EXTERNAL_CONTROLLERS DO
		IF ipExternalControllers[i] <> 0 THEN
			ipExternalControllers[i].StateChanged(_CommandedState);
		END_IF
	END_FOR
END_IF
END_SET
END_PROPERTY

//! @summary Provides fault reaction logic where the module state is driven to the <b>Aborting</b> state
METHOD PROTECTED AbortImmediate

//! @description No error is thrown by this fault reaction.

//! @description This method is called by <c>ComponentMonitor()</c> or <c>SubModuleMonitor()</c> as required
ChangeState(E_PMLCommand.ePMLCommand_Abort);
END_METHOD

//! @summary Provides fault reaction logic where the module state is driven to the <b>Aborting</b> state
METHOD PROTECTED AbortImmediateError
VAR_INPUT
	Name	 : STRING; //! The name of the faulting submodule or component
	IsModule : BOOL;   //! If TRUE a SubModuleError is thrown.  If FALSE a ComponentError is thrown. 
END_VAR

//! @description This fault reaction throws an accompanying error

//! @description This method is called by <c>ComponentMonitor()</c> or <c>SubModuleMonitor()</c> as required
IF IsModule THEN
	IF NOT BaseAlarms[E_BaseAlarms.SubModuleError].bRaised THEN
		F_RaiseAlarmWithStringParameters(BaseAlarms[E_BaseAlarms.SubModuleError],
										 _Name,
										 '',
										 '');
	END_IF
ELSE
	IF NOT BaseAlarms[E_BaseAlarms.ComponentError].bRaised THEN
		F_RaiseAlarmWithStringParameters(BaseAlarms[E_BaseAlarms.ComponentError],
										 _Name,
										 '',
										 '');
	END_IF
END_IF

THIS^.ChangeState(E_PMLCommand.ePMLCommand_Abort);
END_METHOD

//! @summary Provides fault reaction logic where the module state is driven to the <b>Holding</b> state at the next available opportunity
METHOD PROTECTED HoldControlled

(*! <description> No error is thrown by this fault reaction.
	<b> TODO: Needs implementation </b> </description>*)

//! @description This method is called by <c>ComponentMonitor()</c> or <c>SubModuleMonitor()</c> as required
ChangeState(E_PMLCommand.ePMLCommand_Hold);
END_METHOD

//! @summary Provides fault reaction logic where the module state is driven to the <b>Holding</b> state immediately
METHOD PROTECTED HoldImmediate

(*! <description> No error is thrown by this fault reaction.
	<b> TODO: Needs implementation </b> </description>*)

//! @description This method is called by <c>ComponentMonitor()</c> or <c>SubModuleMonitor()</c> as required
ChangeState(E_PMLCommand.ePMLCommand_Hold);
END_METHOD

//! @summary Provides fault reaction logic where the module state is driven to the <b>Stopping</b> state at the next available opportunity
METHOD PROTECTED StopControlled

(*! <description> No error is thrown by this fault reaction.
	<b> TODO: Needs implementation </b> </description>*)

//! @description This method is called by <c>ComponentMonitor()</c> or <c>SubModuleMonitor()</c> as required
ChangeState(E_PMLCommand.ePMLCommand_Stop);
END_METHOD

//! @summary Provides fault reaction logic where the module state is driven to the <b>Stopping</b> state immediately
METHOD PROTECTED StopImmediate

//! @description No error is thrown by this fault reaction.

//! @description This method is called by <c>ComponentMonitor()</c> or <c>SubModuleMonitor()</c> as required
ChangeState(E_PMLCommand.ePMLCommand_Stop);
END_METHOD

//! @summary Provides fault reaction logic where the module state is driven to the <b>Suspending</b> state at the next available opportunity
METHOD PROTECTED SuspendControlled

(*! <description> No error is thrown by this fault reaction.
	<b> TODO: Needs implementation </b> </description>*)

//! @description This method is called by <c>ComponentMonitor()</c> or <c>SubModuleMonitor()</c> as required
ChangeState(E_PMLCommand.ePMLCommand_Suspend);
END_METHOD

//! @summary Provides fault reaction logic where the module state is driven to the <b>Suspending</b> state immediately
METHOD PROTECTED SuspendImmediate

(*! <description> No error is thrown by this fault reaction.
	<b> TODO: Needs implementation </b> </description>*)

//! @description This method is called by <c>ComponentMonitor()</c> or <c>SubModuleMonitor()</c> as required
ChangeState(E_PMLCommand.ePMLCommand_Suspend);
END_METHOD

//! @summary Raises an alarm and passes string arguments as parameters for extra fault context/info
METHOD PROTECTED RaiseAlarmWithStrings
VAR_IN_OUT
	Alarm : FB_TcAlarm; //! Alarm to be raised
END_VAR

VAR_INPUT
	String_1 : STRING; //! First string parameter (The Name of this component will be applied first automatically)
	String_2 : STRING; //! Second string parameter
END_VAR
F_RaiseAlarmWithStringParameters(Alarm	  := Alarm,
								 String_1 := Name,
								 String_2 := String_1,
								 String_3 := String_2);
END_METHOD

//! @summary Sets permissive bit to allow HMI control of module and component functions
METHOD PROTECTED FINAL AllowHMIControl
VAR_INPUT
	ThisModuleOnly : BOOL; //! If TRUE, only the PackML module itself is controllable. If FALSE, all components become controllable as well
END_VAR

VAR
	i : UDINT;
END_VAR

//! @description This method is called as required by the <c>HMIPermissions()</c> method
PackMLBaseModule_HMI.Status.HMIControlAvailable := TRUE;
IF ThisModuleOnly THEN
	FOR i := 1 TO NumberOfComponents DO
		ipComponents[i].BlockHMIControl();
	END_FOR
ELSE
	FOR i := 1 TO NumberOfComponents DO
		ipComponents[i].AllowHMIControl();
	END_FOR
END_IF
END_METHOD

//! @summary Clears permissive bit to disallow HMI control of module and component functions
METHOD PROTECTED FINAL BlockHMIControl
VAR
	i : UDINT;
END_VAR

//! @description This method is called as required by the <c>HMIPermissions()</c> method
PackMLBaseModule_HMI.Status.HMIControlAvailable := FALSE;
FOR i := 1 TO NumberOfComponents DO
	ipComponents[i].BlockHMIControl();
END_FOR
END_METHOD

//! @summary Provides interlocks for HMI control and updates HMI status information for this module
METHOD PROTECTED HMICommunication

//! @description This method is called cyclically by <c>CyclicLogic()</c>
//Extend this method in extended FBs to communicate specific implementation data

//Process HMI requests
HMICommand_RT(CLK := (PackMLBaseModule_HMI.Status.HMIControlAvailable AND NOT HMICommandActive_Descendant) AND
					 (PackMLBaseModule_HMI.Command.ActivateModeLog XOR PackMLBaseModule_HMI.Command.DeactivatModeLog XOR PackMLBaseModule_HMI.Command.ActivateStateLog XOR
					 PackMLBaseModule_HMI.Command.DeactivateStateLog XOR PackMLBaseModule_HMI.Command.Mode <> _CommandedMode XOR PackMLBaseModule_HMI.Command.State <> _CommandedState));

//Desendant components should observe this to interlock HMI commands
HMICommandActive_Base := PackMLBaseModule_HMI.Status.HMIControlAvailable AND
						 (PackMLBaseModule_HMI.Command.ActivateModeLog OR PackMLBaseModule_HMI.Command.DeactivatModeLog OR PackMLBaseModule_HMI.Command.ActivateStateLog OR
						 PackMLBaseModule_HMI.Command.DeactivateStateLog XOR PackMLBaseModule_HMI.Command.Mode <> _CommandedMode XOR PackMLBaseModule_HMI.Command.State <> _CommandedState);

IF HMICommand_RT.Q THEN
	IF PackMLBaseModule_HMI.Command.ActivateModeLog THEN
		_LogModeChanges := TRUE;
	END_IF

	IF PackMLBaseModule_HMI.Command.DeactivatModeLog THEN
		_LogModeChanges := FALSE;
	END_IF

	IF PackMLBaseModule_HMI.Command.ActivateStateLog THEN
		_LogStateChanges := TRUE;
	END_IF

	IF PackMLBaseModule_HMI.Command.DeactivateStateLog THEN
		_LogStateChanges := FALSE;
	END_IF

	IF PackMLBaseModule_HMI.Command.Mode <> _CommandedMode THEN
		ModeCommand := PackMLBaseModule_HMI.Command.Mode;
	END_IF

	IF PackMLBaseModule_HMI.Command.State <> _CommandedState THEN
		StateCommand := PackMLBaseModule_HMI.Command.State;
	END_IF
END_IF

PackMLBaseModule_HMI.Config.Name			:= _Name;
PackMLBaseModule_HMI.Config.LogModeChanges	:= _LogModeChanges;
PackMLBaseModule_HMI.Config.LogStateChanges := _LogStateChanges;
PackMLBaseModule_HMI.Config.ModeNames		:= ModeNames;
PackMLBaseModule_HMI.Status.Mode			:= _CurrentMode;
PackMLBaseModule_HMI.Status.State			:= _CurrentState;
PackMLBaseModule_HMI.Status.Busy			:= _Busy;
PackMLBaseModule_HMI.Status.Error			:= _Error;
PackMLBaseModule_HMI.Status.ErrorID			:= _ErrorID;
END_METHOD

//! @summary Automatically enables and disables HMI control based on the PackML mode
METHOD PROTECTED HMIPermissions

//! @description This method is called cyclically by <c>CyclicLogic()</c>
//General Mode Based Monitoring and handling of HMI control
CASE _CurrentMode OF
	E_PMLUnitMode.ePMLUnitMode_Production:
		CASE _CurrentState OF
			E_PMLState.ePMLState_Stopped:
				AllowHMIControl(ThisModuleOnly := TRUE); //Allow control for recovery
			E_PMLState.ePMLState_Idle:
				BlockHMIControl();

			E_PMLState.ePMLState_Suspended:
				BlockHMIControl();

			E_PMLState.ePMLState_Execute:
				BlockHMIControl();

			E_PMLState.ePMLState_Aborted:
				AllowHMIControl(ThisModuleOnly := TRUE); //Allow control for recovery
			E_PMLState.ePMLState_Held:
				AllowHMIControl(ThisModuleOnly := TRUE); //Allow control for recovery
			E_PMLState.ePMLState_Complete:
				BlockHMIControl();
		END_CASE

	E_PMLUnitMode.ePMLUnitMode_Manual:
		AllowHMIControl(ThisModuleOnly := FALSE);

	E_PMLUnitMode.ePMLUnitMode_Maintenance:
		AllowHMIControl(ThisModuleOnly := FALSE);
END_CASE
END_METHOD

//! @summary This method monitors <b>components</b> within this PackML module and initiates fault responses as required
METHOD PROTECTED ComponentMonitor : BOOL
VAR
	AlarmResponses : ARRAY[0..4] OF E_AlarmResponse; //Temporary response array
	i			   : UDINT;
END_VAR

//! @description This method is called cyclically by <c>CyclicLogic()</c>
FOR i := 1 TO NumberOfComponents DO
	IF _CurrentState <> E_PMLState.ePMLState_Aborted AND _CurrentState <> E_PMLState.ePMLState_Aborting AND _CurrentState <> E_PMLState.ePMLState_Clearing AND
	   _CurrentState <> E_PMLState.ePMLState_Stopped AND _CurrentState <> E_PMLState.ePMLState_Stopping THEN
		AlarmResponses := ipComponents[i].ParentResponseDefinitions;
		CASE AlarmResponses[ipComponents[i].CurrentAlarmSeverity] OF
			E_AlarmResponse.Abort_ImmediateError:
				AbortImmediateError(ipComponents[i].Name, FALSE);

			E_AlarmResponse.Abort_Immediate:
				AbortImmediate();

			E_AlarmResponse.Stop_Immediate:
				StopImmediate();

			E_AlarmResponse.Stop_Controlled:
				StopControlled();

			E_AlarmResponse.Hold_Immediate:
				HoldImmediate();

			E_AlarmResponse.Hold_Controlled:
				HoldControlled();

			E_AlarmResponse.Suspend_Immediate:
				SuspendImmediate();

			E_AlarmResponse.Suspend_Controlled:
				SuspendControlled();

			E_AlarmResponse.NoResponse:
				;
		END_CASE
	ELSIF _CurrentState = E_PMLState.ePMLState_Stopped OR _CurrentState = E_PMLState.ePMLState_Stopping THEN
		AlarmResponses := ipComponents[i].ParentResponseDefinitions;
		CASE AlarmResponses[ipComponents[i].CurrentAlarmSeverity] OF
			E_AlarmResponse.Abort_ImmediateError:
				AbortImmediateError(ipComponents[i].Name, FALSE);

			E_AlarmResponse.Abort_Immediate:
				AbortImmediate();

			E_AlarmResponse.NoResponse:
				;
		END_CASE
	END_IF
END_FOR
END_METHOD

//! @summary This method monitors <b>submodules</b> within this PackML module and initiates fault responses as required
METHOD PROTECTED SubModuleMonitor : BOOL
VAR
	AlarmResponses : ARRAY[0..4] OF E_AlarmResponse; //Temporary response array	
	i			   : UDINT;
END_VAR

//! @description This method is called cyclically by <c>CyclicLogic()</c>
FOR i := 1 TO NumberOfSubModules DO
	IF _CurrentState <> E_PMLState.ePMLState_Aborted AND _CurrentState <> E_PMLState.ePMLState_Aborting AND _CurrentState <> E_PMLState.ePMLState_Clearing AND
	   _CurrentState <> E_PMLState.ePMLState_Stopped AND _CurrentState <> E_PMLState.ePMLState_Stopping THEN
		AlarmResponses := ipSubModules[i].ParentResponseDefinitions;
		CASE AlarmResponses[ipSubModules[i].CurrentAlarmSeverity] OF
			E_AlarmResponse.Abort_ImmediateError:
				AbortImmediateError(ipSubModules[i].Name, TRUE);

			E_AlarmResponse.Abort_Immediate:
				AbortImmediate();

			E_AlarmResponse.Stop_Immediate:
				StopImmediate();

			E_AlarmResponse.Stop_Controlled:
				StopControlled();

			E_AlarmResponse.Hold_Immediate:
				HoldImmediate();

			E_AlarmResponse.Hold_Controlled:
				HoldControlled();

			E_AlarmResponse.Suspend_Immediate:
				SuspendImmediate();

			E_AlarmResponse.Suspend_Controlled:
				SuspendControlled();

			E_AlarmResponse.NoResponse:
				;
		END_CASE
	ELSIF _CurrentState = E_PMLState.ePMLState_Stopped OR _CurrentState = E_PMLState.ePMLState_Stopping THEN
		AlarmResponses := ipSubModules[i].ParentResponseDefinitions;
		CASE AlarmResponses[ipSubModules[i].CurrentAlarmSeverity] OF
			E_AlarmResponse.Abort_ImmediateError:
				AbortImmediateError(ipSubModules[i].Name, TRUE);

			E_AlarmResponse.Abort_Immediate:
				AbortImmediate();

			E_AlarmResponse.NoResponse:
				;
		END_CASE
	END_IF
END_FOR
END_METHOD

//! @summary This method contains code which will execute when this PackML module is in the <b>Aborted</b> state
METHOD PROTECTED Aborted

(*! <description> <b>The base implementation of this method is empty. User must override this method to provide functionality.</b>
<table> 
	<tr>
		<th> Previous State </th>
		<th> Transition In </th>
		<th> Transition Out </th>
		<th> Next State  </th> 
	</tr>
	<tr>
		<td> Aborting </td>
		<td> State Complete <i>(Aborting)</i></td> 
		<td> Clear Command </td>
		<td> Clearing </td> 
	</tr>
</table>
This method is called as required by <c>StateControl()</c>
</description> 

*)
//*************************************************************************************************************************************************************************

//If you are about to write application specific code, note that any such code should exist within the "Application" directory using a Function Block that 'EXTENDS' this base Function Block!

//This particular method's functionality can be overriden in the extended block by creating a method of the same name, with desired functionality therein

//If the functionality of this base module is to be retained, but more functionality is desired, the extended method can contain a SUPER^.ThisMethodName(); call, which will call this code

//*************************************************************************************************************************************************************************
END_METHOD

//! @summary This method contains code which will execute when this PackML module is in the <b>Complete</b> state
METHOD PROTECTED Complete

(*! <description> <b>The base implementation of this method is empty. User must override this method to provide functionality.</b>
<table> 
	<tr>
		<th> Previous State </th>
		<th> Transition In </th>
		<th> Transition Out </th>
		<th> Next State  </th> 
	</tr>
	<tr>
		<td> Completing </td>
		<td> State Complete <i>(Completing)</i></td> 
		<td> Reset Command </td>
		<td> Resetting </td> 
	</tr>
</table>
This method is called as required by <c>StateControl()</c>
</description> 

*)
//*************************************************************************************************************************************************************************

//If you are about to write application specific code, note that any such code should exist within the "Application" directory using a Function Block that 'EXTENDS' this base Function Block!

//This particular method's functionality can be overriden in the extended block by creating a method of the same name, with desired functionality therein

//If the functionality of this base module is to be retained, but more functionality is desired, the extended method can contain a SUPER^.ThisMethodName(); call, which will call this code

//*************************************************************************************************************************************************************************
END_METHOD

//! @summary This method contains code which will execute when this PackML module is in the <b>Execute</b> state
METHOD PROTECTED Execute

(*! <description> <b>The base implementation of this method is empty. User must override this method to provide functionality.</b>
<table> 
	<tr>
		<th> Previous State </th>
		<th> Transition In </th>
		<th> Transition Out </th>
		<th> Next State  </th> 
	</tr>
	<tr>
		<td> Starting<b>-or-</b>Unholding <b>-or-</b>Unsuspending</td>
		<td> State Complete<i>(Starting<b>-or-</b>Unholding<b>-or-</b>Unsuspending)</i></td> 
		<td> State Complete<b>-or-</b>Hold Command<b>-or-</b>Suspend Command</td>
		<td> Completing<b>-or-</b>Holding<b>-or-</b>Suspending</td>
	</tr>
</table>
This method is called as required by <c>StateControl()</c>
</description> 

*)
//*************************************************************************************************************************************************************************

//If you are about to write application specific code, note that any such code should exist within the "Application" directory using a Function Block that 'EXTENDS' this base Function Block!

//This particular method's functionality can be overriden in the extended block by creating a method of the same name, with desired functionality therein

//If the functionality of this base module is to be retained, but more functionality is desired, the extended method can contain a SUPER^.ThisMethodName(); call, which will call this code

//*************************************************************************************************************************************************************************
END_METHOD

//! @summary This method contains code which will execute when this PackML module is in the <b>Held</b> state
METHOD PROTECTED Held

(*! <description> <b>The base implementation of this method is empty. User must override this method to provide functionality.</b>
<table> 
	<tr>
		<th> Previous State </th>
		<th> Transition In </th>
		<th> Transition Out </th>
		<th> Next State  </th> 
	</tr>
	<tr>
		<td> Holding </td>
		<td> State Complete <i>(Holding)</i></td> 
		<td> Unhold Command </td>
		<td> Unholding </td> 
	</tr>
</table>
This method is called as required by <c>StateControl()</c>
</description> 

*)
//*************************************************************************************************************************************************************************

//If you are about to write application specific code, note that any such code should exist within the "Application" directory using a Function Block that 'EXTENDS' this base Function Block!

//This particular method's functionality can be overriden in the extended block by creating a method of the same name, with desired functionality therein

//If the functionality of this base module is to be retained, but more functionality is desired, the extended method can contain a SUPER^.ThisMethodName(); call, which will call this code

//*************************************************************************************************************************************************************************
END_METHOD

//! @summary This method contains code which will execute when this PackML module is in the <b>Idle</b> state
METHOD PROTECTED Idle

(*! <description> <b>The base implementation of this method is empty. User must override this method to provide functionality.</b>
<table> 
	<tr>
		<th> Previous State </th>
		<th> Transition In </th>
		<th> Transition Out </th>
		<th> Next State  </th> 
	</tr>
	<tr>
		<td> Resetting </td>
		<td> State Complete <i>(Resetting)</i></td> 
		<td> Start Command </td>
		<td> Starting </td> 
	</tr>
</table>
This method is called as required by <c>StateControl()</c>
</description> 

*)
//*************************************************************************************************************************************************************************

//If you are about to write application specific code, note that any such code should exist within the "Application" directory using a Function Block that 'EXTENDS' this base Function Block!

//This particular method's functionality can be overriden in the extended block by creating a method of the same name, with desired functionality therein

//If the functionality of this base module is to be retained, but more functionality is desired, the extended method can contain a SUPER^.ThisMethodName(); call, which will call this code

//*************************************************************************************************************************************************************************
END_METHOD

//! @summary This method contains code which will execute when this PackML module is in the <b>Stopped</b> state
METHOD PROTECTED Stopped

(*! <description> <b>The base implementation of this method is empty. User must override this method to provide functionality.</b>
<table> 
	<tr>
		<th> Previous State </th>
		<th> Transition In </th>
		<th> Transition Out </th>
		<th> Next State  </th> 
	</tr>
	<tr>
		<td> Stopping<b>-or-</b>Clearing </td>
		<td> State Complete <i>(Stopping<b>-or-</b>Clearing)</i></td> 
		<td> Reset Command </td>
		<td> Resetting </td> 
	</tr>
</table>
This method is called as required by <c>StateControl()</c>
</description> 

*)
//*************************************************************************************************************************************************************************

//If you are about to write application specific code, note that any such code should exist within the "Application" directory using a Function Block that 'EXTENDS' this base Function Block!

//This particular method's functionality can be overriden in the extended block by creating a method of the same name, with desired functionality therein

//If the functionality of this base module is to be retained, but more functionality is desired, the extended method can contain a SUPER^.ThisMethodName(); call, which will call this code

//*************************************************************************************************************************************************************************
END_METHOD

//! @summary This method contains code which will execute when this PackML module is in the <b>Suspended</b> state
METHOD PROTECTED Suspended

(*! <description> <b>The base implementation of this method is empty. User must override this method to provide functionality.</b>
<table> 
	<tr>
		<th> Previous State </th>
		<th> Transition In </th>
		<th> Transition Out </th>
		<th> Next State  </th> 
	</tr>
	<tr>
		<td> Suspending </td>
		<td> State Complete <i>(Suspending)</i></td> 
		<td> Unsuspend Command </td>
		<td> Unsuspending </td> 
	</tr>
</table>
This method is called as required by <c>StateControl()</c>
</description> 

*)
//*************************************************************************************************************************************************************************

//If you are about to write application specific code, note that any such code should exist within the "Application" directory using a Function Block that 'EXTENDS' this base Function Block!

//This particular method's functionality can be overriden in the extended block by creating a method of the same name, with desired functionality therein

//If the functionality of this base module is to be retained, but more functionality is desired, the extended method can contain a SUPER^.ThisMethodName(); call, which will call this code

//*************************************************************************************************************************************************************************
END_METHOD

//! @summary This method contains code which will execute when this PackML module is in a state which is not defined by the PackML standard
METHOD PROTECTED Undefined

(*! <description> <b>The base implementation of this method is empty. User must override this method to provide functionality.
<i>This state should not be reached under normal circumstances.</i></b>
This method is called as required by <c>StateControl()</c>
</description> 

*)
//*************************************************************************************************************************************************************************

//If you are about to write application specific code, note that any such code should exist within the "Application" directory using a Function Block that 'EXTENDS' this base Function Block!

//This particular method's functionality can be overriden in the extended block by creating a method of the same name, with desired functionality therein

//If the functionality of this base module is to be retained, but more functionality is desired, the extended method can contain a SUPER^.ThisMethodName(); call, which will call this code

//*************************************************************************************************************************************************************************
END_METHOD

//! @summary Handles mode change requests for this module and all submodules
METHOD PRIVATE FINAL ModeControl
VAR
	i : UDINT;
END_VAR

//! @description This method is called cyclically by <c>CyclicLogic()</c>
//On startup, Mode is invalid, set it to production
IF _CurrentMode = E_PMLUnitMode.ePMLUnitMode_Invalid THEN
	ModeChangeRequested := TRUE;
	_CommandedMode		:= Parameters_PackML_Base.UNIT_MODE_DEFAULT;

	//Notify external controllers that state has changed	
	FOR i := 1 TO Parameters_PackML_Base.MAX_NO_OF_EXTERNAL_CONTROLLERS DO
		IF ipExternalControllers[i] <> 0 THEN
			ipExternalControllers[i].ModeChanged(_CommandedMode);
		END_IF
	END_FOR

	LastModeCommand := _CommandedMode;

	//If mode is valid and the command has changed, attempt to change modes
ELSIF _CommandedMode <> LastModeCommand THEN
	ModeChangeRequested				  := TRUE;
	PackMLBaseModule_HMI.Command.Mode := _CommandedMode;

	//Notify external controllers that state has changed	
	FOR i := 1 TO Parameters_PackML_Base.MAX_NO_OF_EXTERNAL_CONTROLLERS DO
		IF ipExternalControllers[i] <> 0 THEN
			ipExternalControllers[i].ModeChanged(_CommandedMode);
		END_IF
	END_FOR

	LastModeCommand := _CommandedMode;
END_IF

IF ModeChangeRequested THEN
	//Handles mode changes based on ModeCommand and the state transition rules defined in the pre-defined protected modes or custom modes
	ModeManager(bExecute	 := TRUE,
				eModeCommand := _CommandedMode,
				eState		 := _CurrentState,
				eModeStatus	 => _CurrentMode);

	IF ModeManager.bDone THEN
		IF PackMLAlarms[E_PackMLBase_Alarms.ModeCommandInvalid].bRaised THEN
			PackMLAlarms[E_PackMLBase_Alarms.ModeCommandInvalid].Clear(0, 0);
		END_IF

		//If PackML mode has changed
		IF ModeManager.eModeStatus <> LastMode THEN
			LastMode				:= ModeManager.eModeStatus;
			SequenceState			:= 0;
			DescendantSequenceState := 0;

			//If state change logging is not suppressed
			IF _LogModeChanges THEN
				PMLModeLogger(Alarms := PackMLAlarms, ModulePrefix := _Name, Mode := ModeManager.eModeStatus);
			END_IF

			// Change SubModules
			FOR i := 1 TO NumberOfSubModules DO
				ipSubModules[i].ModeCommand := ModeManager.eModeStatus; //Call the SetMode loop of the subunits 
			END_FOR
		END_IF

		// Reset mode control command
		ModeManager(bExecute := FALSE);
		ModeChangeRequested := FALSE;
	ELSIF ModeManager.bError THEN
		IF ReachedInitialDefaultStateAndMode THEN
			IF NOT PackMLAlarms[E_PackMLBase_Alarms.ModeCommandInvalid].bRaised THEN
				PackMLAlarms[E_PackMLBase_Alarms.ModeCommandInvalid].Raise(0);
			END_IF
		END_IF

		// Reset mode control command
		ModeManager(bExecute := FALSE);
		ModeChangeRequested := FALSE;
	END_IF
END_IF
END_METHOD

//! @summary Calls PackML state manager and corresponding methods according to current module state
METHOD PRIVATE FINAL StateControl
//! @description This method is called cyclically by <c>CyclicLogic()</c>
VAR
	i : UDINT;
END_VAR
//On startup, state is invalid, set it to default
IF _CurrentState = E_PMLState.ePMLState_Undefined AND _CurrentMode <> E_PMLUnitMode.ePMLUnitMode_Invalid THEN
	_CommandedState := Parameters_PackML_Base.UNIT_STATE_DEFAULT;
END_IF

//Call PackML state machine	
StateMachine(eMode			  := _CurrentMode,
			 eCommand		  := _CommandedState,
			 stSubUnitInfoRef :=,
			 stOptions		  :=,
			 eState			  => _CurrentState,
			 sState			  =>,
			 bError			  =>,
			 nErrorID		  =>);

//If PackML state has changed
IF _CurrentState <> LastState THEN
	LastState						   := _CurrentState;
	PackMLBaseModule_HMI.Command.State := _CommandedState;

	//Notify external controllers that state has changed
	FOR i := 1 TO Parameters_PackML_Base.MAX_NO_OF_EXTERNAL_CONTROLLERS DO
		IF ipExternalControllers[i] <> 0 THEN
			ipExternalControllers[i].StateChanged(_CommandedState);
		END_IF
	END_FOR

	SequenceState			:= 0;
	DescendantSequenceState := 0;
	NoStateTasksToComplete	:= TRUE;
END_IF

IF ReachedInitialDefaultStateAndMode THEN
	//Log appropriate state changes
	PMLStateLogger(Alarms		 := PackMLAlarms,
				   ModulePrefix	 := _Name,
				   State		 := _CurrentState,
				   LogAllChanges := _LogStateChanges);
END_IF

// Call appropriate method depending on current PackML state
CASE _CurrentState OF
	E_PMLState.ePMLState_Undefined:
		Undefined();

	E_PMLState.ePMLState_Clearing:
		Clearing();

	E_PMLState.ePMLState_Stopped:
		Stopped();

	E_PMLState.ePMLState_Starting:
		Starting();

	E_PMLState.ePMLState_Idle:
		Idle();

	E_PMLState.ePMLState_Suspended:
		Suspended();

	E_PMLState.ePMLState_Execute:
		Execute();

	E_PMLState.ePMLState_Stopping:
		Stopping();

	E_PMLState.ePMLState_Aborting:
		Aborting();

	E_PMLState.ePMLState_Aborted:
		Aborted();

	E_PMLState.ePMLState_Holding:
		Holding();

	E_PMLState.ePMLState_Held:
		Held();

	E_PMLState.ePMLState_Unholding:
		Unholding();

	E_PMLState.ePMLState_Suspending:
		Suspending();

	E_PMLState.ePMLState_Unsuspending:
		Unsuspending();

	E_PMLState.ePMLState_Resetting:
		Resetting();

	E_PMLState.ePMLState_Completing:
		Completing();

	E_PMLState.ePMLState_Complete:
		Complete();
END_CASE
END_METHOD

//! @summary This method contains code which will execute when this PackML module is in the <b>Aborting</b> state
METHOD PROTECTED Aborting
VAR
	i				: UDINT;
	SubModulesReady : BOOL := TRUE;
END_VAR

(*! <description> <b>Note:</b> The <i>Abort</i> command should be associated with the fault handing routine of a module. It should not be directly commanded from any user inteface. 

<table> 
	<tr>
		<th> Previous State </th>
		<th> Transition In </th>
		<th> Transition Out </th>
		<th> Next State  </th> 
	</tr>
	<tr>
		<td> <b>ANY</b> </td>
		<td> Abort Command </td> 
		<td> State Complete </td>
		<td> Aborted </td> 
	</tr>
</table>

This method is called as required by <c>StateControl()</c>
</description> 

*)
//*************************************************************************************************************************************************************************

//If you are about to write application specific code, note that any such code should exist within the "Application" directory using a Function Block that 'EXTENDS' this base Function Block!

//This particular method's functionality can be overriden in the extended block by creating a method of the same name, with desired functionality therein

//If the functionality of this base module is to be retained, but more functionality is desired, the extended method can contain a SUPER^.ThisMethodName(); call, which will call this code

//*************************************************************************************************************************************************************************

//Perform State tasks here

// Send abort command to all sub modules
FOR i := 1 TO NumberOfSubModules DO
	ipSubModules[i].StateCommand := ePMLCommand_Abort;
END_FOR

FOR i := 1 TO NumberOfSubModules DO
	SubModulesReady := SubModulesReady AND (ipSubModules[i].CurrentState = ePMLState_Aborted);
END_FOR

IF SubModulesReady AND (StateTasksComplete OR NoStateTasksToComplete) THEN
	NoStateTasksToComplete := TRUE;
	StateTasksComplete	   := FALSE;
	StateComplete();
END_IF
END_METHOD

//! @summary This method contains code which will execute when this PackML module is in the <b>Clearing</b> state
METHOD PROTECTED Clearing
VAR
	i				: UDINT;
	SubModulesReady : BOOL := TRUE;
END_VAR

(*! <description> <b>Note:</b> The <i>Clear</i> command can also be thought of as a <i>fault reset</i> depite the ambiguity in the naming of the <i>Reset</i> state. 
<table> 
	<tr>
		<th> Previous State </th>
		<th> Transition In </th>
		<th> Transition Out </th>
		<th> Next State  </th> 
	</tr>
	<tr>
		<td> Aborted </td>
		<td> Clear Command </td> 
		<td> State Complete </td>
		<td> Stopped </td> 
	</tr>
</table>
This method is called as required by <c>StateControl()</c>
</description> 

*)
//*************************************************************************************************************************************************************************

//If you are about to write application specific code, note that any such code should exist within the "Application" directory using a Function Block that 'EXTENDS' this base Function Block!

//This particular method's functionality can be overriden in the extended block by creating a method of the same name, with desired functionality therein

//If the functionality of this base module is to be retained, but more functionality is desired, the extended method can contain a SUPER^.ThisMethodName(); call, which will call this code

//*************************************************************************************************************************************************************************

//Perform State tasks here

// Send clear command to all sub modules
FOR i := 1 TO NumberOfSubModules DO
	ipSubModules[i].StateCommand := ePMLCommand_Clear;
END_FOR

IF BaseAlarms[E_BaseAlarms.ComponentError].bRaised THEN
	BaseAlarms[E_BaseAlarms.ComponentError].Clear(0, 0);
END_IF;

IF BaseAlarms[E_BaseAlarms.SubModuleError].bRaised THEN
	BaseAlarms[E_BaseAlarms.SubModuleError].Clear(0, 0);
END_IF;

FOR i := 1 TO NumberOfComponents DO
	IF ipComponents[i].Error THEN
		ipComponents[i].Reset();
	END_IF
END_FOR

FOR i := 1 TO NumberOfComponents DO
	SubModulesReady := SubModulesReady AND NOT ipComponents[i].Error;
END_FOR

FOR i := 1 TO NumberOfSubModules DO
	SubModulesReady := SubModulesReady AND (ipSubModules[i].CurrentState = ePMLState_Stopped);
END_FOR

IF SubModulesReady AND (StateTasksComplete OR NoStateTasksToComplete) THEN
	NoStateTasksToComplete := TRUE;
	StateTasksComplete	   := FALSE;
	StateComplete();
END_IF
END_METHOD

//! @summary This method contains code which will execute when this PackML module is in the <b>Completing</b> state
METHOD PROTECTED Completing
VAR
	i				: UDINT;
	SubModulesReady : BOOL := TRUE;
END_VAR

(*! <description><b></b><table> 
	<tr>
		<th> Previous State </th>
		<th> Transition In </th>
		<th> Transition Out </th>
		<th> Next State  </th> 
	</tr>
	<tr>
		<td> Execute </td>
		<td> State Complete <i>(Execute)</i> </td> 
		<td> State Complete </td>
		<td> Completed </td> 
	</tr>
</table>
This method is called as required by <c>StateControl()</c>
</description> 
*)
//*************************************************************************************************************************************************************************

//If you are about to write application specific code, note that any such code should exist within the "Application" directory using a Function Block that 'EXTENDS' this base Function Block!

//This particular method's functionality can be overriden in the extended block by creating a method of the same name, with desired functionality therein

//If the functionality of this base module is to be retained, but more functionality is desired, the extended method can contain a SUPER^.ThisMethodName(); call, which will call this code

//*************************************************************************************************************************************************************************

//Perform State tasks here

// Send complete command to all sub modules
FOR i := 1 TO NumberOfSubModules DO
	ipSubModules[i].StateCommand := ePMLCommand_Complete;
END_FOR

FOR i := 1 TO NumberOfSubModules DO
	SubModulesReady := SubModulesReady AND (ipSubModules[i].CurrentState = ePMLState_Complete);
END_FOR

IF SubModulesReady AND (StateTasksComplete OR NoStateTasksToComplete) THEN
	NoStateTasksToComplete := TRUE;
	StateTasksComplete	   := FALSE;
	StateComplete();
END_IF
END_METHOD

//! @summary This method contains code which will execute when this PackML module is in the <b>Holding</b> state
METHOD PROTECTED Holding
VAR
	i				: UDINT;
	SubModulesReady : BOOL := TRUE;
END_VAR

(*! <description><b>Note:</b> The <i>Hold</i> command is intended to be given by an operator. It is meant to be distinct from a <i>Suspend</i> in that upstream/downstream jams, etc. should be handled automatically using <i>Suspend</i>.  Both <i>Hold</i>and<i>Suspend</i> result in a <i>paused</i> state which should allow resumption of the <b>Execute</b> state. 
<table> 
	<tr>
		<th> Previous State </th>
		<th> Transition In </th>
		<th> Transition Out </th>
		<th> Next State  </th> 
	</tr>
	<tr>
		<td> Execute </td>
		<td> Hold Command </td> 
		<td> State Complete </td>
		<td> Held </td> 
	</tr>
</table>
This method is called as required by <c>StateControl()</c>
</description> 

*)
//*************************************************************************************************************************************************************************

//If you are about to write application specific code, note that any such code should exist within the "Application" directory using a Function Block that 'EXTENDS' this base Function Block!

//This particular method's functionality can be overriden in the extended block by creating a method of the same name, with desired functionality therein

//If the functionality of this base module is to be retained, but more functionality is desired, the extended method can contain a SUPER^.ThisMethodName(); call, which will call this code

//*************************************************************************************************************************************************************************

//Perform State tasks here

// Send hold command to all sub modules
FOR i := 1 TO NumberOfSubModules DO
	ipSubModules[i].StateCommand := ePMLCommand_Hold;
END_FOR

FOR i := 1 TO NumberOfSubModules DO
	SubModulesReady := SubModulesReady AND (ipSubModules[i].CurrentState = ePMLState_Held);
END_FOR

IF SubModulesReady AND (StateTasksComplete OR NoStateTasksToComplete) THEN
	NoStateTasksToComplete := TRUE;
	StateTasksComplete	   := FALSE;
	StateComplete();
END_IF
END_METHOD

//! @summary This method contains code which will execute when this PackML module is in the <b>Resetting</b> state
METHOD PROTECTED Resetting
VAR
	i				: UDINT;
	SubModulesReady : BOOL := TRUE;
END_VAR

(*! <description> <b>Note:</b> The <i>Reset</i> command can also be thought of as an <i>enable</i> depite the ambiguity in the naming of the <i>Clearing</i> state.
<table> 
	<tr>
		<th> Previous State </th>
		<th> Transition In </th>
		<th> Transition Out </th>
		<th> Next State  </th> 
	</tr>
	<tr>
		<td> Stopped<b>-or-</b>Completed </td>
		<td> Reset Command </td> 
		<td> State Complete </td>
		<td> Idle </td> 
	</tr>
</table>
This method is called as required by <c>StateControl()</c>
</description> 

*)
//*************************************************************************************************************************************************************************

//If you are about to write application specific code, note that any such code should exist within the "Application" directory using a Function Block that 'EXTENDS' this base Function Block!

//This particular method's functionality can be overriden in the extended block by creating a method of the same name, with desired functionality therein

//If the functionality of this base module is to be retained, but more functionality is desired, the extended method can contain a SUPER^.ThisMethodName(); call, which will call this code

//*************************************************************************************************************************************************************************

//Perform State tasks here

// Send clear/reset command to all sub modules

//As long as this module is in the "Resetting" state, it will attempt to get all modules to Idle by sending abort, clear, and reset commands as appropriate to its children until they do
FOR i := 1 TO NumberOfSubModules DO
	IF ipSubModules[i].CurrentState = ePMLState_Stopped OR ipSubModules[i].CurrentState = ePMLState_Complete THEN
		ipSubModules[i].StateCommand := ePMLCommand_Reset;
	ELSIF ipSubModules[i].CurrentState = ePMLState_Aborted THEN
		ipSubModules[i].StateCommand := ePMLCommand_Clear;
	ELSIF ipSubModules[i].CurrentState = ePMLState_Clearing OR ipSubModules[i].CurrentState = ePMLState_Stopping OR ipSubModules[i].CurrentState = ePMLState_Resetting OR
		  ipSubModules[i].CurrentState = ePMLState_Idle THEN
		;
	ELSE
		ipSubModules[i].StateCommand := ePMLCommand_Abort;
	END_IF
END_FOR

FOR i := 1 TO NumberOfSubModules DO
	SubModulesReady := SubModulesReady AND (ipSubModules[i].CurrentState = ePMLState_Idle);
END_FOR

IF SubModulesReady AND (StateTasksComplete OR NoStateTasksToComplete) THEN
	NoStateTasksToComplete := TRUE;
	StateTasksComplete	   := FALSE;
	StateComplete();
END_IF
END_METHOD

//! @summary This method contains code which will execute when this PackML module is in the <b>Starting</b> state
METHOD PROTECTED Starting
VAR
	i				: UDINT;
	SubModulesReady : BOOL := TRUE;
END_VAR

(*! <description><b></b><table> 
	<tr>
		<th> Previous State </th>
		<th> Transition In </th>
		<th> Transition Out </th>
		<th> Next State  </th> 
	</tr>
	<tr>
		<td> Idle </td>
		<td> Start Command </td> 
		<td> State Complete </td>
		<td> Execute </td> 
	</tr>
</table>
This method is called as required by <c>StateControl()</c>
</description> 

*)
//*************************************************************************************************************************************************************************

//If you are about to write application specific code, note that any such code should exist within the "Application" directory using a Function Block that 'EXTENDS' this base Function Block!

//This particular method's functionality can be overriden in the extended block by creating a method of the same name, with desired functionality therein

//If the functionality of this base module is to be retained, but more functionality is desired, the extended method can contain a SUPER^.ThisMethodName(); call, which will call this code

//*************************************************************************************************************************************************************************

//Perform State tasks here

// Send start command to all sub modules
FOR i := 1 TO NumberOfSubModules DO
	ipSubModules[i].StateCommand := ePMLCommand_Start;
END_FOR

FOR i := 1 TO NumberOfSubModules DO
	SubModulesReady := SubModulesReady AND (ipSubModules[i].CurrentState = ePMLState_Execute);
END_FOR

IF SubModulesReady AND (StateTasksComplete OR NoStateTasksToComplete) THEN
	NoStateTasksToComplete := TRUE;
	StateTasksComplete	   := FALSE;
	StateComplete();
END_IF
END_METHOD

//! @summary This method contains code which will execute when this PackML module is in the <b>Stopping</b> state
METHOD PROTECTED Stopping
VAR
	i				: UDINT;
	SubModulesReady : BOOL := TRUE;
END_VAR

(*! <description><b></b><table> 
	<tr>
		<th> Previous State </th>
		<th> Transition In </th>
		<th> Transition Out </th>
		<th> Next State  </th> 
	</tr>
	<tr>
		<td> <b>ANY<i>except</i></b>Stopped<b>-or-</b>Clearing<b>-or-</b>Aborted<b>-or-</b>Aborting</td>
		<td> Stop Command </td> 
		<td> State Complete </td>
		<td> Stopped </td> 
	</tr>
</table>
This method is called as required by <c>StateControl()</c>
</description> 

*)
//*************************************************************************************************************************************************************************

//If you are about to write application specific code, note that any such code should exist within the "Application" directory using a Function Block that 'EXTENDS' this base Function Block!

//This particular method's functionality can be overriden in the extended block by creating a method of the same name, with desired functionality therein

//If the functionality of this base module is to be retained, but more functionality is desired, the extended method can contain a SUPER^.ThisMethodName(); call, which will call this code

//*************************************************************************************************************************************************************************

//Perform State tasks here

// Send stop command to all sub modules
FOR i := 1 TO NumberOfSubModules DO
	ipSubModules[i].StateCommand := ePMLCommand_Stop;
END_FOR

FOR i := 1 TO NumberOfSubModules DO
	SubModulesReady := SubModulesReady AND (ipSubModules[i].CurrentState = ePMLState_Stopped OR ipSubModules[i].CurrentState = ePMLState_Aborted);
END_FOR

IF SubModulesReady AND (StateTasksComplete OR NoStateTasksToComplete) THEN
	NoStateTasksToComplete := TRUE;
	StateTasksComplete	   := FALSE;
	StateComplete();
END_IF
END_METHOD

//! @summary This method contains code which will execute when this PackML module is in the <b>Suspending</b> state
METHOD PROTECTED Suspending
VAR
	i				: UDINT;
	SubModulesReady : BOOL := TRUE;
END_VAR

(*! <description><b>Note:</b> The <i>Suspend</i> command is intended to be initiated by automatic detection of upstream/downstream jams, etc. It is meant to be distinct from a <i>Hold</i> in that <i>Hold</i> should be commanded by an operator.  Both <i>Hold</i>and<i>Suspend</i> result in a <i>paused</i> state which should allow resumption of the <b>Execute</b> state. 
<table> 
	<tr>
		<th> Previous State </th>
		<th> Transition In </th>
		<th> Transition Out </th>
		<th> Next State  </th> 
	</tr>
	<tr>
		<td> Execute </td>
		<td> Suspend Command </td> 
		<td> State Complete </td>
		<td> Suspended </td> 
	</tr>
</table>
This method is called as required by <c>StateControl()</c>
</description> 

*)
//*************************************************************************************************************************************************************************

//If you are about to write application specific code, note that any such code should exist within the "Application" directory using a Function Block that 'EXTENDS' this base Function Block!

//This particular method's functionality can be overriden in the extended block by creating a method of the same name, with desired functionality therein

//If the functionality of this base module is to be retained, but more functionality is desired, the extended method can contain a SUPER^.ThisMethodName(); call, which will call this code

//*************************************************************************************************************************************************************************

//Perform State tasks here

// Send suspend command to all sub modules
FOR i := 1 TO NumberOfSubModules DO
	ipSubModules[i].StateCommand := ePMLCommand_Suspend;
END_FOR

FOR i := 1 TO NumberOfSubModules DO
	SubModulesReady := SubModulesReady AND (ipSubModules[i].CurrentState = ePMLState_Suspended);
END_FOR

IF SubModulesReady AND (StateTasksComplete OR NoStateTasksToComplete) THEN
	NoStateTasksToComplete := TRUE;
	StateTasksComplete	   := FALSE;
	StateComplete();
END_IF
END_METHOD

//! @summary This method contains code which will execute when this PackML module is in the <b>Unholding</b> state
METHOD PROTECTED Unholding
VAR
	i				: UDINT;
	SubModulesReady : BOOL := TRUE;
END_VAR

(*! <description><b></b><table> 
	<tr>
		<th> Previous State </th>
		<th> Transition In </th>
		<th> Transition Out </th>
		<th> Next State  </th> 
	</tr>
	<tr>
		<td> Held </td>
		<td> Unhold Command </td> 
		<td> State Complete </td>
		<td> Execute </td> 
	</tr>
</table>
This method is called as required by <c>StateControl()</c>
</description> 

*)
//*************************************************************************************************************************************************************************

//If you are about to write application specific code, note that any such code should exist within the "Application" directory using a Function Block that 'EXTENDS' this base Function Block!

//This particular method's functionality can be overriden in the extended block by creating a method of the same name, with desired functionality therein

//If the functionality of this base module is to be retained, but more functionality is desired, the extended method can contain a SUPER^.ThisMethodName(); call, which will call this code

//*************************************************************************************************************************************************************************

//Perform State tasks here

// Send unhold command to all sub modules
FOR i := 1 TO NumberOfSubModules DO
	ipSubModules[i].StateCommand := ePMLCommand_Unhold;
END_FOR

FOR i := 1 TO NumberOfSubModules DO
	SubModulesReady := SubModulesReady AND (ipSubModules[i].CurrentState = ePMLState_Execute);
END_FOR

IF SubModulesReady AND (StateTasksComplete OR NoStateTasksToComplete) THEN
	NoStateTasksToComplete := TRUE;
	StateTasksComplete	   := FALSE;
	StateComplete();
END_IF
END_METHOD

//! @summary This method contains code which will execute when this PackML module is in the <b>Unsuspending</b> state
METHOD PROTECTED Unsuspending
VAR
	i				: UDINT;
	SubModulesReady : BOOL := TRUE;
END_VAR

(*! <description><b></b><table> 
	<tr>
		<th> Previous State </th>
		<th> Transition In </th>
		<th> Transition Out </th>
		<th> Next State  </th> 
	</tr>
	<tr>
		<td> Suspended </td>
		<td> Unsuspend Command </td> 
		<td> State Complete </td>
		<td> Execute </td> 
	</tr>
</table>
This method is called as required by <c>StateControl()</c>
</description> 

*)
//*************************************************************************************************************************************************************************

//If you are about to write application specific code, note that any such code should exist within the "Application" directory using a Function Block that 'EXTENDS' this base Function Block!

//This particular method's functionality can be overriden in the extended block by creating a method of the same name, with desired functionality therein

//If the functionality of this base module is to be retained, but more functionality is desired, the extended method can contain a SUPER^.ThisMethodName(); call, which will call this code

//*************************************************************************************************************************************************************************

//Perform State tasks here

// Send unsuspend command to all sub modules
FOR i := 1 TO NumberOfSubModules DO
	ipSubModules[i].StateCommand := ePMLCommand_Unsuspend;
END_FOR

FOR i := 1 TO NumberOfSubModules DO
	SubModulesReady := SubModulesReady AND (ipSubModules[i].CurrentState = ePMLState_Execute);
END_FOR

IF SubModulesReady AND (StateTasksComplete OR NoStateTasksToComplete) THEN
	NoStateTasksToComplete := TRUE;
	StateTasksComplete	   := FALSE;
	StateComplete();
END_IF
END_METHOD

//! @summary Initializes event function blocks using this module's name
{attribute 'call_after_online_change_slot' := '<slot>'}
METHOD PROTECTED CreateEvents

//! @description This method is called by <c>Initialize()</c> as required
F_CreateAllEventsInClass(Alarms		:= PackMLAlarms,
						 ClassSize	:= SIZEOF(TC_EVENTS.PackMLBase_Alarms),
						 pInitEvent := ADR(TC_EVENTS.PackMLBase_Alarms.InitReferenceEvent),
						 Prefix		:= _Name);

F_CreateAllEventsInClass(Alarms		:= BaseAlarms,
						 ClassSize	:= SIZEOF(TC_EVENTS.BaseAlarms),
						 pInitEvent := ADR(TC_EVENTS.BaseAlarms.InitReferenceEvent),
						 Prefix		:= _Name);
END_METHOD

//! @summary Basic module initialization logic
METHOD PROTECTED Initialize : BOOL;
VAR
	i						 : UDINT;
	varInfo					 : __SYSTEM.VAR_INFO;
	AllSubUnitsInitialized	 : BOOL := TRUE;
	AllComponentsInitialized : BOOL := TRUE;
END_VAR

//! @description This method is called by <c>CyclicLogic()</c> as required
//This method may get called several times while waiting for subunits/components to init

//so it makes sense to break it up into a state machine
CASE SequenceState OF
	0:
		CreateEvents();
		SequenceState := SequenceState + 10;

	10:
		// Figure out how many Submodules were instantiated - they should be from 1 to X and not skip any indices.
		NumberOfSubModules := 0;
		FOR i := 1 TO Parameters_PackML_Base.MAX_NO_OF_SUBMODULES DO
			IF ipSubModules[i] <> 0 THEN
				NumberOfSubModules		   := NumberOfSubModules + 1;
				PMLSubModuleInfo[i].Active := TRUE; // Follows Main State Machine
			END_IF
		END_FOR

		SequenceState := SequenceState + 10;

	20:
		NumberOfComponents := 0;
		FOR i := 1 TO Parameters_PackML_Base.MAX_NO_OF_COMPONENTS DO
			IF ipComponents[i] <> 0 THEN
				NumberOfComponents	 := NumberOfComponents + 1;
				ipComponents[i].Name := CONCAT(CONCAT(_Name, ' '), ipComponents[i].Name); //Add the name of the module as a prefix to the name given in the declaration initialization
			END_IF
		END_FOR

		SequenceState := SequenceState + 10;

	30:
		// Initialize subunit overview used by state machine
		PMLSubModuleInfoRef.ArraySize	 := SIZEOF(PMLSubModuleInfo);
		PMLSubModuleInfoRef.NoOfSubUnits := NumberOfSubModules;
		PMLSubModuleInfoRef.pArray		 := ADR(PMLSubModuleInfo);
		SequenceState					 := SequenceState + 10;

	40:
		// Initialization for this module is not complete until all subunits/components are finished

		// with their own Initialize().  This is called from CyclicLogic() so call from here until they are initialized.
		FOR i := 1 TO NumberOfSubModules DO
			IF ipSubModules[i] <> 0 AND_THEN NOT ipSubModules[i].InitComplete THEN
				AllSubUnitsInitialized := FALSE;
				ipSubModules[i].CyclicLogic();
			END_IF
		END_FOR

		FOR i := 1 TO NumberOfComponents DO
			IF ipComponents[i] <> 0 AND_THEN NOT ipComponents[i].InitComplete THEN
				AllComponentsInitialized := FALSE;
				ipComponents[i].CyclicLogic();
			END_IF
		END_FOR

		IF AllSubUnitsInitialized AND AllComponentsInitialized THEN
			SequenceState := 0;
			Initialize	  := TRUE;
		END_IF
END_CASE
END_METHOD

METHOD PROTECTED FINAL RegisterComponent
VAR_INPUT
	Component : I_ComponentBase;
END_VAR

VAR
	i		: UDINT;
	PLCStop : PLC_Stop;
END_VAR
IF NOT _InitComplete AND (Component <> 0) THEN
	FOR i := 1 TO SPT_BaseTypes.Parameters_PackML_Base.MAX_NO_OF_COMPONENTS DO
		IF ipComponents[i] = Component THEN
			//Component already registered
			RETURN;
		END_IF
	END_FOR	



	FOR i := 1 TO SPT_BaseTypes.Parameters_PackML_Base.MAX_NO_OF_COMPONENTS DO
		IF ipComponents[i] = 0 THEN
			ipComponents[i] := Component;
			RETURN;
		END_IF
	END_FOR

	//If we get here then we are exceeding the array bounds
	Trace(CONCAT('***CRITICAL - Failed to register component!!  (', CONCAT(Component.Name, ')***')));
	PLCStop(STOP := TRUE);
END_IF
END_METHOD

METHOD FINAL RegisterExternalController : BOOL
VAR_INPUT
	Controller : I_PackML_ExternalController;
END_VAR

VAR
	i : UDINT;
END_VAR
FOR i := 1 TO Parameters_PackML_Base.MAX_NO_OF_EXTERNAL_CONTROLLERS DO
	IF ipExternalControllers[i] = 0 THEN
		ipExternalControllers[i]   := Controller;
		Controller.Control		   := THIS^;
		RegisterExternalController := TRUE;
		RETURN;
	END_IF
END_FOR

//If you get this far you have already registered the maximum number of controllers
RegisterExternalController := FALSE;
END_METHOD

METHOD PROTECTED FINAL RegisterSubmodule
VAR_INPUT
	SubModule : I_PackML_BaseModule;
END_VAR

VAR
	i		: UDINT;
	PLCStop : PLC_Stop;
END_VAR
IF NOT _InitComplete AND (SubModule <> 0) THEN
	FOR i := 1 TO SPT_BaseTypes.Parameters_PackML_Base.MAX_NO_OF_SUBMODULES DO
		IF ipSubModules[i] = SubModule THEN
			//Submodule already registered
			RETURN;
		END_IF
	END_FOR	



	FOR i := 1 TO SPT_BaseTypes.Parameters_PackML_Base.MAX_NO_OF_SUBMODULES DO
		IF ipSubModules[i] = 0 THEN
			ipSubModules[i] := SubModule;
			RETURN;
		END_IF
	END_FOR

	//If we get here then we are exceeding the array bounds
	Trace(CONCAT('***CRITICAL - Failed to register SubModule!!  (', CONCAT(SubModule.Name, ')***')));
	PLCStop(STOP := TRUE);
END_IF
END_METHOD

//! @summary Signals to the state manager FB when a state has completed
METHOD PROTECTED StateComplete

//! @description This method is called by any of the transition state's logic methods (<c>...<b>ing()</b></c>) as required
//*************************************************************************************************************************************************************************

//If you are about to write application specific code, note that any such code should exist within the "Application" directory using a Function Block that 'EXTENDS' this base Function Block!

//This particular method's functionality can be overriden in the extended block by creating a method of the same name, with desired functionality therein

//If the functionality of this base module is to be retained, but more functionality is desired, the extended method can contain a SUPER^.ThisMethodName(); call, which will call this code

//*************************************************************************************************************************************************************************
StateMachine.M_StateComplete();
END_METHOD

END_FUNCTION_BLOCK

// PackML/FB_PackML_StateLogger
//! @summary This FB raises events corresponding to <b>state</b> changes within the parent PackML module
FUNCTION_BLOCK FB_PackML_StateLogger
VAR_IN_OUT
	Alarms : ARRAY[1..48] OF FB_TcAlarm; //! Array of alarms for Core PackML events that exist in any PackML enabled module
END_VAR

VAR_INPUT
	ModulePrefix  : STRING;		  //! Prefix String for all state change events (Typically the ID and Name of the module in some concatenated form) <TODO> Remove this? </TODO>
	State		  : E_PMLState;	  //! Current PackML state of the module
	LogAllChanges : BOOL := TRUE; //! If TRUE, all state change events will be logged, regardless of severity, otherwise info alarms are ignored
END_VAR

VAR
	LastState  : E_PMLState := E_PMLState.ePMLState_Aborted; //Saves the previous state each time the block is run
	pTempAlarm : REFERENCE TO FB_TcAlarm;					 //Temporary reference that makes severity checking simpler vs individually checking each change alarm within the case statement
END_VAR

IF State <> LastState THEN //If state has changed
	CASE State OF		   //Get the stored alarm that corresponds to the newly entered state and save its reference temporarily
		E_PMLState.ePMLState_Starting:
			pTempAlarm REF= Alarms[E_PackMLBase_Alarms.StateStartingEnter];

		E_PMLState.ePMLState_Execute:
			pTempAlarm REF= Alarms[E_PackMLBase_Alarms.StateExecuteEnter];

		E_PMLState.ePMLState_Completing:
			pTempAlarm REF= Alarms[E_PackMLBase_Alarms.StateCompletingEnter];

		E_PMLState.ePMLState_Complete:
			pTempAlarm REF= Alarms[E_PackMLBase_Alarms.StateCompleteEnter];

		E_PMLState.ePMLState_Resetting:
			pTempAlarm REF= Alarms[E_PackMLBase_Alarms.StateResettingEnter];

		E_PMLState.ePMLState_Idle:
			pTempAlarm REF= Alarms[E_PackMLBase_Alarms.StateIdleEnter];

		E_PMLState.ePMLState_Holding:
			pTempAlarm REF= Alarms[E_PackMLBase_Alarms.StateHoldingEnter];

		E_PMLState.ePMLState_Held:
			pTempAlarm REF= Alarms[E_PackMLBase_Alarms.StateHeldEnter];

		E_PMLState.ePMLState_Unholding:
			pTempAlarm REF= Alarms[E_PackMLBase_Alarms.StateUnholdingEnter];

		E_PMLState.ePMLState_Suspending:
			pTempAlarm REF= Alarms[E_PackMLBase_Alarms.StateSuspendingEnter];

		E_PMLState.ePMLState_Suspended:
			pTempAlarm REF= Alarms[E_PackMLBase_Alarms.StateSuspendedEnter];

		E_PMLState.ePMLState_Unsuspending:
			pTempAlarm REF= Alarms[E_PackMLBase_Alarms.StateUnsuspendingEnter];

		E_PMLState.ePMLState_Stopping:
			pTempAlarm REF= Alarms[E_PackMLBase_Alarms.StateStoppingEnter];

		E_PMLState.ePMLState_Stopped:
			pTempAlarm REF= Alarms[E_PackMLBase_Alarms.StateStoppedEnter];

		E_PMLState.ePMLState_Aborting:
			pTempAlarm REF= Alarms[E_PackMLBase_Alarms.StateAbortingEnter];

		E_PMLState.ePMLState_Aborted:
			pTempAlarm REF= Alarms[E_PackMLBase_Alarms.StateAbortedEnter];

		E_PMLState.ePMLState_Clearing:
			pTempAlarm REF= Alarms[E_PackMLBase_Alarms.StateClearingEnter];

		E_PMLState.ePMLState_Undefined:
			pTempAlarm REF= Alarms[E_PackMLBase_Alarms.StateUndefinedEnter];
	END_CASE

	//If the FB is set to log all changes, log the change, otherwise check the severity of the alarm and log it if it exceeds 'info' severity
	IF LogAllChanges OR (pTempAlarm.eSeverity <> TcEventSeverity.Info AND pTempAlarm.eSeverity <> TcEventSeverity.Verbose) THEN
		pTempAlarm.Raise(0);
	END_IF

	CASE LastState OF //Clear the previous state's event (Events will remain 'Raised' as long as the module remains in that state)
		E_PMLState.ePMLState_Starting:
			Alarms[E_PackMLBase_Alarms.StateStartingEnter].Clear(0, 0);

		E_PMLState.ePMLState_Execute:
			Alarms[E_PackMLBase_Alarms.StateExecuteEnter].Clear(0, 0);

		E_PMLState.ePMLState_Completing:
			Alarms[E_PackMLBase_Alarms.StateCompletingEnter].Clear(0, 0);

		E_PMLState.ePMLState_Complete:
			Alarms[E_PackMLBase_Alarms.StateCompleteEnter].Clear(0, 0);

		E_PMLState.ePMLState_Resetting:
			Alarms[E_PackMLBase_Alarms.StateResettingEnter].Clear(0, 0);

		E_PMLState.ePMLState_Idle:
			Alarms[E_PackMLBase_Alarms.StateIdleEnter].Clear(0, 0);

		E_PMLState.ePMLState_Holding:
			Alarms[E_PackMLBase_Alarms.StateHoldingEnter].Clear(0, 0);

		E_PMLState.ePMLState_Held:
			Alarms[E_PackMLBase_Alarms.StateHeldEnter].Clear(0, 0);

		E_PMLState.ePMLState_Unholding:
			Alarms[E_PackMLBase_Alarms.StateUnholdingEnter].Clear(0, 0);

		E_PMLState.ePMLState_Suspending:
			Alarms[E_PackMLBase_Alarms.StateSuspendingEnter].Clear(0, 0);

		E_PMLState.ePMLState_Suspended:
			Alarms[E_PackMLBase_Alarms.StateSuspendedEnter].Clear(0, 0);

		E_PMLState.ePMLState_Unsuspending:
			Alarms[E_PackMLBase_Alarms.StateUnsuspendingEnter].Clear(0, 0);

		E_PMLState.ePMLState_Stopping:
			Alarms[E_PackMLBase_Alarms.StateStoppingEnter].Clear(0, 0);

		E_PMLState.ePMLState_Stopped:
			Alarms[E_PackMLBase_Alarms.StateStoppedEnter].Clear(0, 0);

		E_PMLState.ePMLState_Aborting:
			Alarms[E_PackMLBase_Alarms.StateAbortingEnter].Clear(0, 0);

		E_PMLState.ePMLState_Aborted:
			Alarms[E_PackMLBase_Alarms.StateAbortedEnter].Clear(0, 0);

		E_PMLState.ePMLState_Clearing:
			Alarms[E_PackMLBase_Alarms.StateClearingEnter].Clear(0, 0);

		E_PMLState.ePMLState_Undefined:
			Alarms[E_PackMLBase_Alarms.StateUndefinedEnter].Clear(0, 0);
	END_CASE

	LastState := State; //Store previous state
END_IF

(*! <description> The current state is compared against the mode during the last call.  The corresponding events are raised/cleared as the state is changed.
<b>This FB is called from FB_PMLModuleBase.StateControl.  Further calls are not necessary.</b></description>*)

END_FUNCTION_BLOCK

// PackML/FB_PackML_ModeLogger
//! @summary This FB raises events corresponding to <b>mode</b> changes within the parent PackML module
FUNCTION_BLOCK FB_PackML_ModeLogger
VAR_IN_OUT
	Alarms : ARRAY[1..48] OF FB_TcAlarm; //! Array of alarms for Core PackML events that exist in any PackML enabled module
END_VAR

VAR_INPUT
	ModulePrefix : STRING; //! Prefix String for any  <TODO> Remove this? </TODO>
	Mode		 : DINT;   //! Current mode of the module
END_VAR

VAR
	LastMode : DINT;
END_VAR

IF Mode <> LastMode THEN
	CASE Mode OF
		E_PMLUnitMode.ePMLUnitMode_Invalid:
			Alarms[E_PackMLBase_Alarms.ModeInvalidEnter].Raise(0);

		E_PMLUnitMode.ePMLUnitMode_Production:
			Alarms[E_PackMLBase_Alarms.ModeProductionEnter].Raise(0);

		E_PMLUnitMode.ePMLUnitMode_Maintenance:
			Alarms[E_PackMLBase_Alarms.ModeMaintenanceEnter].Raise(0);

		E_PMLUnitMode.ePMLUnitMode_Manual:
			Alarms[E_PackMLBase_Alarms.ModeManualEnter].Raise(0);
	END_CASE

	CASE LastMode OF
		E_PMLUnitMode.ePMLUnitMode_Invalid:
			Alarms[E_PackMLBase_Alarms.ModeInvalidEnter].Clear(0, 0);

		E_PMLUnitMode.ePMLUnitMode_Production:
			Alarms[E_PackMLBase_Alarms.ModeProductionEnter].Clear(0, 0);

